fbStateSetup(stPositionState:=fbIM1K1.stOut, fPosition:=-8.82, sPmpsState:='IM1K1:PPM-OUT');
fbStateSetup(stPositionState:=fbIM1K1.stPower, fPosition:=-47.92, sPmpsState:='IM1K1:PPM-POWERMETER');
fbStateSetup(stPositionState:=fbIM1K1.stYag1, fPosition:=-71.92, sPmpsState:='IM1K1:PPM-YAG1');
fbStateSetup(stPositionState:=fbIM1K1.stYag2, fPosition:=-97.93, sPmpsState:='IM1K1:PPM-YAG2');

fbIM1K1(
    fbFFHWO := GVL.fbFastFaultOutput1,
    fbArbiter := GVL.fbArbiter1,
    stYStage := Main.M1,
    sDeviceName := 'IM1K1:PPM',
    sTransitionKey := 'IM1K1:PPM-TRANSITION',
    bEnableMotion := TRUE,
    bEnableBeamParams := TRUE,
    bEnablePositionLimits := TRUE,
    fResponsivity := 0.0624,
);

END_PROGRAM

// ---- POUs/PRG_IM2K1_PPM.TcPOU
PROGRAM PRG_IM2K1_PPM
VAR
    {attribute 'pytmc' := 'pv: IM2K1:PPM'}
    {attribute 'TcLinkTo' := '.fbGige.iIlluminatorINT := TIIB[IM2K1-EL4004]^AO Outputs Channel 1^Analog output;
                              .fbGige.bGigePower := TIIB[IM2K1-EL2004]^Channel 2^Output;
                              .fbPowerMeter.iVoltageINT := TIIB[IM2K1-EL3062]^AI Standard Channel 1^Value;
                              .fbPowerMeter.fbTempSensor.bError := TIIB[IM2K1-EL3314]^TC Inputs Channel 1^Status^Error;
                              .fbPowerMeter.fbTempSensor.bUnderrange := TIIB[IM2K1-EL3314]^TC Inputs Channel 1^Status^Underrange;
                              .fbPowerMeter.fbTempSensor.bOverrange := TIIB[IM2K1-EL3314]^TC Inputs Channel 1^Status^Overrange;
                              .fbPowerMeter.fbTempSensor.iRaw := TIIB[IM2K1-EL3314]^TC Inputs Channel 1^Value;
                              .fbYagTempSensor.bError := TIIB[IM2K1-EL3314]^TC Inputs Channel 2^Status^Error;
                              .fbYagTempSensor.bUnderrange := TIIB[IM2K1-EL3314]^TC Inputs Channel 2^Status^Underrange;
                              .fbYagTempSensor.bOverrange := TIIB[IM2K1-EL3314]^TC Inputs Channel 2^Status^Overrange;
                              .fbYagTempSensor.iRaw := TIIB[IM2K1-EL3314]^TC Inputs Channel 2^Value'}
    fbIM2K1: FB_PPM;

    fbStateSetup: FB_StateSetupHelper;
    stDefault: ST_PositionState := (
        fVelocity := 13,
        bMoveOk := TRUE,
        bValid := TRUE
    );
END_VAR


fbStateSetup(stPositionState:=stDefault, bSetDefault:=TRUE);

fbStateSetup(stPositionState:=fbIM2K1.stOut, fPosition:=-9.09, sPmpsState:='IM2K1:PPM-OUT');
fbStateSetup(stPositionState:=fbIM2K1.stPower, fPosition:=-48.19, sPmpsState:='IM2K1:PPM-POWERMETER');
fbStateSetup(stPositionState:=fbIM2K1.stYag1, fPosition:=-72.19, sPmpsState:='IM2K1:PPM-YAG1');
fbStateSetup(stPositionState:=fbIM2K1.stYag2, fPosition:=-98.2, sPmpsState:='IM2K1:PPM-YAG2');

fbIM2K1(
    fbFFHWO := GVL.fbFastFaultOutput1,
    fbArbiter := GVL.fbArbiter1,
    stYStage := Main.M2,
    sDeviceName := 'IM2K1:PPM',
    sTransitionKey := 'IM2K1:PPM-TRANSITION',
    bEnableMotion := TRUE,
    bEnableBeamParams := TRUE,
    bEnablePositionLimits := TRUE,
    fResponsivity := 0.0625,
);

END_PROGRAM

// ---- POUs/PRG_IM1K2_PPM.TcPOU
PROGRAM PRG_IM1K2_PPM
VAR
    {attribute 'pytmc' := 'pv: IM1K2:PPM'}
    {attribute 'TcLinkTo' := '.fbGige.iIlluminatorINT := TIIB[IM1K2-EL4004-E7]^AO Outputs Channel 1^Analog output;
                              .fbGige.bGigePower := TIIB[IM1K2-EL2004-E3]^Channel 2^Output;
                              .fbPowerMeter.iVoltageINT := TIIB[IM1K2-EL3062-E6]^AI Standard Channel 1^Value;
                              .fbPowerMeter.fbTempSensor.bError := TIIB[IM1K2-EL3314-E4]^TC Inputs Channel 1^Status^Error;
                              .fbPowerMeter.fbTempSensor.bUnderrange := TIIB[IM1K2-EL3314-E4]^TC Inputs Channel 1^Status^Underrange;
                              .fbPowerMeter.fbTempSensor.bOverrange := TIIB[IM1K2-EL3314-E4]^TC Inputs Channel 1^Status^Overrange;
                              .fbPowerMeter.fbTempSensor.iRaw := TIIB[IM1K2-EL3314-E4]^TC Inputs Channel 1^Value;
                              .fbYagTempSensor.bError := TIIB[IM1K2-EL3314-E4]^TC Inputs Channel 2^Status^Error;
                              .fbYagTempSensor.bUnderrange := TIIB[IM1K2-EL3314-E4]^TC Inputs Channel 2^Status^Underrange;
                              .fbYagTempSensor.bOverrange := TIIB[IM1K2-EL3314-E4]^TC Inputs Channel 2^Status^Overrange;
                              .fbYagTempSensor.iRaw := TIIB[IM1K2-EL3314-E4]^TC Inputs Channel 2^Value;
                              .fbFlowMeter.iRaw := TIIB[IM1K2-EL3052-E5]^AI Standard Channel 1^Value'}
    fbIM1K2: FB_PPM;

    fbStateSetup: FB_StateSetupHelper;
    stDefault: ST_PositionState := (
        fVelocity := 12,
        bMoveOk := TRUE,
        bValid := TRUE
    );
END_VAR


fbStateSetup(stPositionState:=stDefault, bSetDefault:=TRUE);

fbStateSetup(stPositionState:=fbIM1K2.stOut, fPosition:=-9.82, sPmpsState:='IM1K2:PPM-OUT');
fbStateSetup(stPositionState:=fbIM1K2.stPower, fPosition:=-48.92, sPmpsState:='IM1K2:PPM-POWERMETER');
fbStateSetup(stPositionState:=fbIM1K2.stYag1, fPosition:=-72.92, sPmpsState:='IM1K2:PPM-YAG1');
fbStateSetup(stPositionState:=fbIM1K2.stYag2, fPosition:=-98.93, sPmpsState:='IM1K2:PPM-YAG2');

fbIM1K2(
    fbFFHWO := GVL.fbFastFaultOutput1,
    fbArbiter := GVL.fbArbiter1,
    stYStage := Main.M4,
    sDeviceName := 'IM1K2:PPM',
    sTransitionKey := 'IM1K2:PPM-TRANSITION',
    bEnableMotion := TRUE,
    bEnableBeamParams := TRUE,
    bEnablePositionLimits := TRUE,
    fResponsivity := 0.0513,
);

END_PROGRAM

// ---- POUs/PRG_AL1K2_L2SI.TcPOU
PROGRAM PRG_AL1K2_L2SI
VAR
    {attribute 'pytmc' := 'pv: AL1K2:L2SI'}
    {attribute 'TcLinkTo' := '.fbLaser.iLaserINT := TIIB[AL1K2-EL4004-E4]^AO Outputs Channel 1^Analog output;
                              .fbLaser.iShutdownINT := TIIB[AL1K2-EL4004-E4]^AO Outputs Channel 2^Analog output'}
    fbAL1K2: FB_REF;

    fbStateSetup: FB_StateSetupHelper;
    stDefault: ST_PositionState := (
        fVelocity := 10,
        bMoveOk := TRUE,
        bValid := TRUE
    );
END_VAR


fbStateSetup(stPositionState:=stDefault, bSetDefault:=TRUE);

fbStateSetup(stPositionState:=fbAL1K2.stOut, fPosition:=-33.5, sPmpsState:='AL1K2:L2SI-OUT');
fbStateSetup(stPositionState:=fbAL1K2.stIn, fPosition:=-75, sPmpsState:='AL1K2:L2SI-IN');

fbAL1K2(
    fbFFHWO := GVL.fbFastFaultOutput2,
    fbArbiter := GVL.fbArbiter2,
    stYStage := Main.M5,
    sDeviceName := 'AL1K2:L2SI',
    sTransitionKey := 'AL1K2:L2SI-TRANSITION',
    bEnableMotion := TRUE,
    bEnableBeamParams := TRUE,
    bEnablePositionLimits := TRUE,
);

END_PROGRAM

// ---- POUs/PRG_IM2K2_PPM.TcPOU
PROGRAM PRG_IM2K2_PPM
VAR
    {attribute 'pytmc' := 'pv: IM2K2:PPM'}
    {attribute 'TcLinkTo' := '.fbGige.iIlluminatorINT := TIIB[IM2K2-EL4004-E7]^AO Outputs Channel 1^Analog output;
                              .fbGige.bGigePower := TIIB[IM2K2-EL2004-E3]^Channel 2^Output;
                              .fbPowerMeter.iVoltageINT := TIIB[IM2K2-EL3062-E6]^AI Standard Channel 1^Value;
                              .fbPowerMeter.fbTempSensor.bError := TIIB[IM2K2-EL3314-E4]^TC Inputs Channel 1^Status^Error;
                              .fbPowerMeter.fbTempSensor.bUnderrange := TIIB[IM2K2-EL3314-E4]^TC Inputs Channel 1^Status^Underrange;
                              .fbPowerMeter.fbTempSensor.bOverrange := TIIB[IM2K2-EL3314-E4]^TC Inputs Channel 1^Status^Overrange;
                              .fbPowerMeter.fbTempSensor.iRaw := TIIB[IM2K2-EL3314-E4]^TC Inputs Channel 1^Value;
                              .fbYagTempSensor.bError := TIIB[IM2K2-EL3314-E4]^TC Inputs Channel 2^Status^Error;
                              .fbYagTempSensor.bUnderrange := TIIB[IM2K2-EL3314-E4]^TC Inputs Channel 2^Status^Underrange;
                              .fbYagTempSensor.bOverrange := TIIB[IM2K2-EL3314-E4]^TC Inputs Channel 2^Status^Overrange;
                              .fbYagTempSensor.iRaw := TIIB[IM2K2-EL3314-E4]^TC Inputs Channel 2^Value;
                              .fbFlowMeter.iRaw := TIIB[IM1K2-EL3052-E5]^AI Standard Channel 1^Value'}
// IM2K2 shares the same flow meter as IM1K2
    fbIM2K2: FB_PPM;

    fbStateSetup: FB_StateSetupHelper;
    stDefault: ST_PositionState := (
        fVelocity := 15,
        bMoveOk := TRUE,
        bValid := TRUE
    );
END_VAR


fbStateSetup(stPositionState:=stDefault, bSetDefault:=TRUE);

fbStateSetup(stPositionState:=fbIM2K2.stOut, fPosition:=-8.49, sPmpsState:='IM2K2:PPM-OUT');
fbStateSetup(stPositionState:=fbIM2K2.stPower, fPosition:=-47.59, sPmpsState:='IM2K2:PPM-POWERMETER');
fbStateSetup(stPositionState:=fbIM2K2.stYag1, fPosition:=-71.59, sPmpsState:='IM2K2:PPM-YAG1');
fbStateSetup(stPositionState:=fbIM2K2.stYag2, fPosition:=-97.60, sPmpsState:='IM2K2:PPM-YAG2');

fbIM2K2(
    fbFFHWO := GVL.fbFastFaultOutput2,
    fbArbiter := GVL.fbArbiter2,
    stYStage := Main.M6,
    sDeviceName := 'IM2K2:PPM',
    sTransitionKey := 'IM2K2:PPM-TRANSITION',
    bEnableMotion := TRUE,
    bEnableBeamParams := TRUE,
    bEnablePositionLimits := TRUE,
    fResponsivity := 0.0670,
);

END_PROGRAM

// ---- POUs/PRG_IM3K2_PPM.TcPOU
PROGRAM PRG_IM3K2_PPM
VAR
    {attribute 'pytmc' := 'pv: IM3K2:PPM'}
    {attribute 'TcLinkTo' := '.fbGige.iIlluminatorINT := TIIB[IM3K2-EL4004-E7]^AO Outputs Channel 1^Analog output;
                              .fbGige.bGigePower := TIIB[IM3K2-EL2004-E3]^Channel 2^Output;
                              .fbPowerMeter.iVoltageINT := TIIB[IM3K2-EL3062-E6]^AI Standard Channel 1^Value;
                              .fbPowerMeter.fbTempSensor.bError := TIIB[IM3K2-EL3314-E4]^TC Inputs Channel 1^Status^Error;
                              .fbPowerMeter.fbTempSensor.bUnderrange := TIIB[IM3K2-EL3314-E4]^TC Inputs Channel 1^Status^Underrange;
                              .fbPowerMeter.fbTempSensor.bOverrange := TIIB[IM3K2-EL3314-E4]^TC Inputs Channel 1^Status^Overrange;
                              .fbPowerMeter.fbTempSensor.iRaw := TIIB[IM3K2-EL3314-E4]^TC Inputs Channel 1^Value;
                              .fbYagTempSensor.bError := TIIB[IM3K2-EL3314-E4]^TC Inputs Channel 2^Status^Error;
                              .fbYagTempSensor.bUnderrange := TIIB[IM3K2-EL3314-E4]^TC Inputs Channel 2^Status^Underrange;
                              .fbYagTempSensor.bOverrange := TIIB[IM3K2-EL3314-E4]^TC Inputs Channel 2^Status^Overrange;
                              .fbYagTempSensor.iRaw := TIIB[IM3K2-EL3314-E4]^TC Inputs Channel 2^Value;
                              .fbFlowMeter.iRaw := TIIB[IM1K2-EL3052-E5]^AI Standard Channel 1^Value'}
// IM3K2 shares the same flow meter as IM1K2
    fbIM3K2: FB_PPM;

    fbStateSetup: FB_StateSetupHelper;
    stDefault: ST_PositionState := (
        fVelocity := 14,
        bMoveOk := TRUE,
        bValid := TRUE
    );
END_VAR


fbStateSetup(stPositionState:=stDefault, bSetDefault:=TRUE);

fbStateSetup(stPositionState:=fbIM3K2.stOut, fPosition:=-9.61, sPmpsState:='IM3K2:PPM-OUT');
fbStateSetup(stPositionState:=fbIM3K2.stPower, fPosition:=-48.71, sPmpsState:='IM3K2:PPM-POWERMETER');
fbStateSetup(stPositionState:=fbIM3K2.stYag1, fPosition:=-72.71, sPmpsState:='IM3K2:PPM-YAG1');
fbStateSetup(stPositionState:=fbIM3K2.stYag2, fPosition:=-98.72, sPmpsState:='IM3K2:PPM-YAG2');

fbIM3K2(
    fbFFHWO := GVL.fbFastFaultOutput2,
    fbArbiter := GVL.fbArbiter2,
    stYStage := Main.M7,
    sDeviceName := 'IM3K2:PPM',
    sTransitionKey := 'IM3K2:PPM-TRANSITION',
    bEnableMotion := TRUE,
    bEnableBeamParams := TRUE,
    bEnablePositionLimits := TRUE,
    fResponsivity := 0.0503
);

END_PROGRAM

// ---- POUs/PRG_IM4K2_PPM.TcPOU
PROGRAM PRG_IM4K2_PPM
VAR
    {attribute 'pytmc' := 'pv: IM4K2:PPM'}
    {attribute 'TcLinkTo' := '.fbGige.iIlluminatorINT := TIIB[IM4K2-EL4004-E7]^AO Outputs Channel 1^Analog output;
                              .fbGige.bGigePower := TIIB[IM4K2-EL2004-E3]^Channel 2^Output;
                              .fbPowerMeter.iVoltageINT := TIIB[IM4K2-EL3602-0002-E8]^AI Inputs Channel 1^Value;
                              .fbPowerMeter.fbTempSensor.bError := TIIB[IM4K2-EL3314-E4]^TC Inputs Channel 1^Status^Error;
                              .fbPowerMeter.fbTempSensor.bUnderrange := TIIB[IM4K2-EL3314-E4]^TC Inputs Channel 1^Status^Underrange;
                              .fbPowerMeter.fbTempSensor.bOverrange := TIIB[IM4K2-EL3314-E4]^TC Inputs Channel 1^Status^Overrange;
                              .fbPowerMeter.fbTempSensor.iRaw := TIIB[IM4K2-EL3314-E4]^TC Inputs Channel 1^Value;
                              .fbYagTempSensor.bError := TIIB[IM4K2-EL3314-E4]^TC Inputs Channel 2^Status^Error;
                              .fbYagTempSensor.bUnderrange := TIIB[IM4K2-EL3314-E4]^TC Inputs Channel 2^Status^Underrange;
                              .fbYagTempSensor.bOverrange := TIIB[IM4K2-EL3314-E4]^TC Inputs Channel 2^Status^Overrange;
                              .fbYagTempSensor.iRaw := TIIB[IM4K2-EL3314-E4]^TC Inputs Channel 2^Value;
                              .fbFlowMeter.iRaw := TIIB[IM1K2-EL3052-E5]^AI Standard Channel 1^Value'}
// IM4K2 shares the same flow meter as IM1K2
    fbIM4K2: FB_PPM;

    fbStateSetup: FB_StateSetupHelper;
    stDefault: ST_PositionState := (
        fVelocity := 12,
        bMoveOk := TRUE,
        bValid := TRUE
    );
END_VAR


fbStateSetup(stPositionState:=stDefault, bSetDefault:=TRUE);

fbStateSetup(stPositionState:=fbIM4K2.stOut, fPosition:=-10.80, sPmpsState:='IM4K2:PPM-OUT');
fbStateSetup(stPositionState:=fbIM4K2.stPower, fPosition:=-49.90, sPmpsState:='IM4K2:PPM-POWERMETER');
fbStateSetup(stPositionState:=fbIM4K2.stYag1, fPosition:=-73.90, sPmpsState:='IM4K2:PPM-YAG1');
fbStateSetup(stPositionState:=fbIM4K2.stYag2, fPosition:=-99.91, sPmpsState:='IM4K2:PPM-YAG2');

fbIM4K2(
    fbFFHWO := GVL.fbFastFaultOutput2,
    fbArbiter := GVL.fbArbiter2,
    stYStage := Main.M8,
    sDeviceName := 'IM4K2:PPM',
    sTransitionKey := 'IM4K2:PPM-TRANSITION',
    bEnableMotion := TRUE,
    bEnableBeamParams := TRUE,
    bEnablePositionLimits := TRUE,
    fResponsivity := 0.0584,
    iTermBits := 31,
    fTermMax := 200,
    fTermMin := 0,
);

END_PROGRAM

// ---- POUs/PRG_TM1K2_ATM.TcPOU
PROGRAM PRG_TM1K2_ATM
VAR
    {attribute 'pytmc' := 'pv: TM1K2:ATM'}
    {attribute 'TcLinkTo' := '.fbThermoCouple1.bError := TIIB[TM1K2-EL3314-E5]^TC Inputs Channel 1^Status^Error;
                              .fbThermoCouple1.bUnderrange := TIIB[TM1K2-EL3314-E5]^TC Inputs Channel 1^Status^Underrange;
                              .fbThermoCouple1.bOverrange := TIIB[TM1K2-EL3314-E5]^TC Inputs Channel 1^Status^Overrange;
                              .fbThermoCouple1.iRaw := TIIB[TM1K2-EL3314-E5]^TC Inputs Channel 1^Value;
                              .fbFlowMeter.iRaw := TIIB[AT1K2-EL3052-E8]^AI Standard Channel 1^Value

'} // TM1K2 shares the same cooling meter as AT1K2
    fbTM1K2: FB_TM1K2;

    fbStateSetup: FB_StateSetupHelper;
    stDefault: ST_PositionState := (
        fVelocity := 1,
        bMoveOk := TRUE,
        bValid := TRUE
    );
END_VAR


fbStateSetup(stPositionState:=stDefault, bSetDefault:=TRUE);

fbStateSetup(stPositionState:=fbTM1K2.stOut, fPosition:=-16.00, fDelta:=7, sPmpsState:='TM1K2:ATM-OUT');
fbStateSetup(stPositionState:=fbTM1K2.stTarget1, fPosition:=-28, fDelta:=7, sPmpsState:='TM1K2:ATM-TARGET1');
fbStateSetup(stPositionState:=fbTM1K2.stTarget2, fPosition:=-38, fDelta:=7, sPmpsState:='TM1K2:ATM-TARGET2');
fbStateSetup(stPositionState:=fbTM1K2.stTarget3, fPosition:=-48, fDelta:=7, sPmpsState:='TM1K2:ATM-TARGET3');
fbStateSetup(stPositionState:=fbTM1K2.stTarget4, fPosition:=-58, fDelta:=7, sPmpsState:='TM1K2:ATM-TARGET4');
fbStateSetup(stPositionState:=fbTM1K2.stTarget5, fPosition:=-68, fDelta:=7, sPmpsState:='TM1K2:ATM-TARGET5');
fbStateSetup(stPositionState:=fbTM1K2.stTarget6, fPosition:=-80, fDelta:=7, sPmpsState:='TM1K2:ATM-TARGET6');
fbStateSetup(stPositionState:=fbTM1K2.stTarget7, fPosition:=-96, fDelta:=7, sPmpsState:='TM1K2:ATM-TARGET7');
fbStateSetup(stPositionState:=fbTM1K2.stTarget8, fPosition:=-114.5, fDelta:=7, sPmpsState:='TM1K2:ATM-TARGET8');

fbTM1K2(
    fbFFHWO := GVL.fbFastFaultOutput2,
    fbArbiter := GVL.fbArbiter2,
    stYStage := Main.M9,
    stXStage := Main.M10,
    sDeviceName := 'TM1K2:ATM',
    sTransitionKey := 'TM1K2:ATM-TRANSITION',
    bEnableMotion := TRUE,
    bEnableBeamParams := TRUE,
    bEnablePositionLimits := TRUE,
);

END_PROGRAM

// ---- POUs/TM1K2/FB_TM1K2.TcPOU
FUNCTION_BLOCK FB_TM1K2
(*
    Function block for Arrival Time Monitor (ATM) controls:
    - X, Y motion
    - Y target states
    - thermocouple

    For TM1K2, we make the following adjustments:
    - Add stTarget6 to the inputs
    - Change the array pragma from 1..6 to 1..7 (1 out and 6 in states, up from 5 in states)
    - Use E_TM1K2_States instead of E_ATM_States

    Add array to 1..9
*)
VAR_IN_OUT
    // Y motor (state select).
    stYStage: ST_MotionStage;
    // X motor (align target to beam).
    stXStage: ST_MotionStage;
    // The fast fault output to fault to.
    fbFFHWO: FB_HardwareFFOutput;
    // The arbiter to request beam conditions from.
    fbArbiter: FB_Arbiter;
END_VAR
VAR_INPUT
    // Settings for the OUT state.
    stOut: ST_PositionState;
    // Settings for the TARGET1 state.
    stTarget1: ST_PositionState;
    // Settings for the TARGET2 state.
    stTarget2: ST_PositionState;
    // Settings for the TARGET3 state.
    stTarget3: ST_PositionState;
    // Settings for the TARGET4 state.
    stTarget4: ST_PositionState;
    // Settings for the TARGET5 state.
    stTarget5: ST_PositionState;
    // Settings for the TARGET6 state.
    stTarget6: ST_PositionState;
    // Settings for the TARGET7 state.
    stTarget7: ST_PositionState;
    // Settings for the TARGET8 state.
    stTarget8: ST_PositionState;
    // Set this to a non-unknown value to request a new move.
    {attribute 'pytmc' := '
        pv: MMS:STATE:SET
        io: io
    '}
    eEnumSet: E_TM1K2_States;
    // Set this to TRUE to enable input state moves, or FALSE to disable them.
    bEnableMotion: BOOL;
    // Set this to TRUE to enable beam parameter checks, or FALSE to disable them.
    bEnableBeamParams: BOOL;
    // Set this to TRUE to enable position limit checks, or FALSE to disable them.
    bEnablePositionLimits: BOOL;
    // The name of the device for use in the PMPS DB lookup and diagnostic screens.
    sDeviceName: STRING;
    // The name of the transition state in the PMPS database.
    sTransitionKey: STRING;
    // Set this to TRUE to re-read the loaded database immediately (useful for debug).
    bReadDBNow: BOOL;
END_VAR
VAR_OUTPUT
    // The current position state as an enum.
    {attribute 'pytmc' := '
        pv: MMS:STATE:GET
        io: i
    '}
    eEnumGet: E_TM1K2_States;
    // The PMPS database lookup associated with the current position state.
    stDbStateParams: ST_DbStateParams;
END_VAR
VAR
    bInit: BOOL;

    fbYStage: FB_MotionStage;
    fbXStage: FB_MotionStage;

    fbStateDefaults: FB_PositionState_Defaults;

    {attribute 'pytmc' := '
        pv: MMS
        astPositionState.array: 1..7
    '}
    fbStates: FB_PositionStatePMPS1D;
    astPositionState: ARRAY[1..GeneralConstants.MAX_STATES] OF ST_PositionState;
    fbArrCheckWrite: FB_CheckPositionStateWrite;

    {attribute 'pytmc' := 'pv: STC:01'}
    fbThermoCouple1: FB_TempSensor;

    {attribute 'pytmc' :='pv: FWM'}
    fbFlowMeter: FB_AnalogInput := (iTermBits:=15, fTermMax:=60, fTermMin:=0);
END_VAR
VAR CONSTANT
    // State defaults if not provided
    fDelta: LREAL := 2;
    fAccel: LREAL := 200;
    fOutDecel: LREAL := 25;
END_VAR


IF NOT bInit THEN
    bInit := TRUE;

    stYStage.nEnableMode := E_StageEnableMode.DURING_MOTION;
    stXStage.nEnableMode := E_StageEnableMode.DURING_MOTION;

    // Partial backcompat, this used to set fVelocity too but this should be set per install
    fbStateDefaults(stPositionState:=stOut, sNameDefault:='OUT', fDeltaDefault:=fDelta, fAccelDefault:=fAccel, fDecelDefault:=fOutDecel);
    fbStateDefaults(stPositionState:=stTarget1, sNameDefault:='TARGET1', fDeltaDefault:=fDelta, fAccelDefault:=fAccel, fDecelDefault:=fAccel);
    fbStateDefaults(stPositionState:=stTarget2, sNameDefault:='TARGET2', fDeltaDefault:=fDelta, fAccelDefault:=fAccel, fDecelDefault:=fAccel);
    fbStateDefaults(stPositionState:=stTarget3, sNameDefault:='TARGET3', fDeltaDefault:=fDelta, fAccelDefault:=fAccel, fDecelDefault:=fAccel);
    fbStateDefaults(stPositionState:=stTarget4, sNameDefault:='TARGET4', fDeltaDefault:=fDelta, fAccelDefault:=fAccel, fDecelDefault:=fAccel);
    fbStateDefaults(stPositionState:=stTarget5, sNameDefault:='TARGET5', fDeltaDefault:=fDelta, fAccelDefault:=fAccel, fDecelDefault:=fAccel);
    fbStateDefaults(stPositionState:=stTarget6, sNameDefault:='TARGET6', fDeltaDefault:=fDelta, fAccelDefault:=fAccel, fDecelDefault:=fAccel);
    fbStateDefaults(stPositionState:=stTarget7, sNameDefault:='TARGET7', fDeltaDefault:=fDelta, fAccelDefault:=fAccel, fDecelDefault:=fAccel);
    fbStateDefaults(stPositionState:=stTarget8, sNameDefault:='TARGET8', fDeltaDefault:=fDelta, fAccelDefault:=fAccel, fDecelDefault:=fAccel);
END_IF

stYStage.bHardwareEnable := TRUE;
stYStage.bPowerSelf := FALSE;

stXStage.bLimitForwardEnable := TRUE;
stXStage.bLimitBackwardEnable := TRUE;
stXStage.bHardwareEnable := TRUE;
stXStage.bPowerSelf := TRUE;

fbYStage(stMotionStage:=stYStage);
fbXStage(stMotionStage:=stXStage);

// We need to update from PLC or from EPICS, but not both
fbArrCheckWrite(
    astPositionState:=astPositionState,
    bCheck:=TRUE,
    bSave:=FALSE,
);
IF NOT fbArrCheckWrite.bHadWrite THEN
    astPositionState[E_TM1K2_States.OUT] := stOut;
    astPositionState[E_TM1K2_States.TARGET1] := stTarget1;
    astPositionState[E_TM1K2_States.TARGET2] := stTarget2;
    astPositionState[E_TM1K2_States.TARGET3] := stTarget3;
    astPositionState[E_TM1K2_States.TARGET4] := stTarget4;
    astPositionState[E_TM1K2_States.TARGET5] := stTarget5;
    astPositionState[E_TM1K2_States.TARGET6] := stTarget6;
    astPositionState[E_TM1K2_States.TARGET7] := stTarget7;
    astPositionState[E_TM1K2_States.TARGET8] := stTarget8;
END_IF

fbStates(
    stMotionStage:=stYStage,
    astPositionState:=astPositionState,
    eEnumSet:=eEnumSet,
    eEnumGet:=eEnumGet,
    fbFFHWO:=fbFFHWO,
    fbArbiter:=fbArbiter,
    bEnableMotion:=bEnableMotion,
    bEnableBeamParams:=bEnableBeamParams,
    bEnablePositionLimits:=bEnablePositionLimits,
    sDeviceName:=sDeviceName,
    sTransitionKey:=sTransitionKey,
    bReadDBNow:=bReadDBNow,
    stDbStateParams=>stDbStateParams,
);

fbArrCheckWrite(
    astPositionState:=astPositionState,
    bCheck:=FALSE,
    bSave:=TRUE,
);

stOut := astPositionState[E_TM1K2_States.OUT];
stTarget1 := astPositionState[E_TM1K2_States.TARGET1];
stTarget2 := astPositionState[E_TM1K2_States.TARGET2];
stTarget3 := astPositionState[E_TM1K2_States.TARGET3];
stTarget4 := astPositionState[E_TM1K2_States.TARGET4];
stTarget5 := astPositionState[E_TM1K2_States.TARGET5];
stTarget6 := astPositionState[E_TM1K2_States.TARGET6];
stTarget7 := astPositionState[E_TM1K2_States.TARGET7];
stTarget8 := astPositionState[E_TM1K2_States.TARGET8];

fbThermoCouple1();
fbFlowMeter();

END_FUNCTION_BLOCK

// ---- POUs/PRG_LI2K2_K2A.TcPOU
PROGRAM PRG_LI2K2_K2A
VAR
    {attribute 'pytmc' := 'pv: LI2K2:K2A'}
    fbLI2K2: FB_LIC;

    fbStateSetup: FB_StateSetupHelper;
    stDefault: ST_PositionState := (
        fVelocity := 1,
        bMoveOk := TRUE,
        bValid := TRUE
    );
END_VAR


fbStateSetup(stPositionState:=stDefault, bSetDefault:=TRUE);

fbStateSetup(stPositionState:=fbLI2K2.stOut, fPosition:=1.2, sPmpsState:='LI2K2:K2A-OUT');
fbStateSetup(stPositionState:=fbLI2K2.stMirror1, fPosition:=-35.3, sPmpsState:='LI2K2:K2A-MIRROR1');
fbStateSetup(stPositionState:=fbLI2K2.stMirror2, fPosition:=-69.3, sPmpsState:='LI2K2:K2A-MIRROR2');
fbStateSetup(stPositionState:=fbLI2K2.stTarget1, fPosition:=-101.3, sPmpsState:='LI2K2:K2A-TARGET1');

fbLI2K2(
    fbFFHWO := GVL.fbFastFaultOutput2,
    fbArbiter := GVL.fbArbiter2,
    stYStage := Main.M11,
    sDeviceName := 'LI2K2:K2A',
    sTransitionKey := 'LI2K2:K2A-TRANSITION',
    bEnableMotion := TRUE,
    bEnableBeamParams := TRUE,
    bEnablePositionLimits := TRUE,
);

END_PROGRAM

// ---- POUs/PRG_PF1K2_WFS.TcPOU
PROGRAM PRG_PF1K2_WFS
VAR
    {attribute 'pytmc' := 'pv: PF1K2:WFS'}
    {attribute 'TcLinkTo' := '.fbThermoCouple1.bError 		:= TIIB[PF1K2-EL3314-E5]^TC Inputs Channel 1^Status^Error;
                              .fbThermoCouple1.bUnderrange	:= TIIB[PF1K2-EL3314-E5]^TC Inputs Channel 1^Status^Underrange;
                              .fbThermoCouple1.bOverrange 	:= TIIB[PF1K2-EL3314-E5]^TC Inputs Channel 1^Status^Overrange;
                              .fbThermoCouple1.iRaw 		:= TIIB[PF1K2-EL3314-E5]^TC Inputs Channel 1^Value;
                              .fbThermoCouple2.bError 		:= TIIB[PF1K2-EL3314-E5]^TC Inputs Channel 2^Status^Error;
                              .fbThermoCouple2.bUnderrange 	:= TIIB[PF1K2-EL3314-E5]^TC Inputs Channel 2^Status^Underrange;
                              .fbThermoCouple2.bOverrange 	:= TIIB[PF1K2-EL3314-E5]^TC Inputs Channel 2^Status^Overrange;
                              .fbThermoCouple2.iRaw 		:= TIIB[PF1K2-EL3314-E5]^TC Inputs Channel 2^Value;
                              .fbFlowMeter.iRaw := TIIB[IM5K2-EL3052-E5]^AI Standard Channel 1^Value

'} // PF1K2 shares the same flow meter as IM5K2
    fbPF1K2: FB_WFS;

    fbStateSetup: FB_StateSetupHelper;
    stDefault: ST_PositionState := (
        fVelocity := 1,
        bMoveOk := TRUE,
        bValid := TRUE
    );
END_VAR


fbStateSetup(stPositionState:=stDefault, bSetDefault:=TRUE);

fbStateSetup(stPositionState:=fbPF1K2.stOut, fPosition:=-13.80, sPmpsState:='PF1K2:WFS-OUT');
fbStateSetup(stPositionState:=fbPF1K2.stTarget1, fPosition:=-94.00, sPmpsState:='PF1K2:WFS-TARGET1');
fbStateSetup(stPositionState:=fbPF1K2.stTarget2, fPosition:=-82.755, sPmpsState:='PF1K2:WFS-TARGET2');
fbStateSetup(stPositionState:=fbPF1K2.stTarget3, fPosition:=-68.38, sPmpsState:='PF1K2:WFS-TARGET3');
fbStateSetup(stPositionState:=fbPF1K2.stTarget4, fPosition:=-54.004, sPmpsState:='PF1K2:WFS-TARGET4');
fbStateSetup(stPositionState:=fbPF1K2.stTarget5, fPosition:=-39.629, sPmpsState:='PF1K2:WFS-TARGET5');

fbPF1K2(
    fbFFHWO := GVL.fbFastFaultOutput2,
    fbArbiter := GVL.fbArbiter2,
    stYStage := Main.M12,
    stZStage := Main.M13,
    sDeviceName := 'PF1K2:WFS',
    sTransitionKey := 'PF1K2:WFS-TRANSITION',
    bEnableMotion := TRUE,
    bEnableBeamParams := TRUE,
    bEnablePositionLimits := TRUE,
    eEnumGet=>GVL.ePF1K2State,
);

END_PROGRAM

// ---- POUs/PRG_IM5K2_PPM.TcPOU
PROGRAM PRG_IM5K2_PPM
VAR
    {attribute 'pytmc' := 'pv: IM5K2:PPM'}
    {attribute 'TcLinkTo' := '.fbGige.iIlluminatorINT := TIIB[IM5K2-EL4004-E7]^AO Outputs Channel 1^Analog output;
                              .fbGige.bGigePower := TIIB[IM5K2-EL2004-E3]^Channel 2^Output;
                              .fbPowerMeter.iVoltageINT := TIIB[IM5K2-EL3062-E6]^AI Standard Channel 1^Value;
                              .fbPowerMeter.fbTempSensor.bError := TIIB[IM5K2-EL3314-E4]^TC Inputs Channel 1^Status^Error;
                              .fbPowerMeter.fbTempSensor.bUnderrange := TIIB[IM5K2-EL3314-E4]^TC Inputs Channel 1^Status^Underrange;
                              .fbPowerMeter.fbTempSensor.bOverrange := TIIB[IM5K2-EL3314-E4]^TC Inputs Channel 1^Status^Overrange;
                              .fbPowerMeter.fbTempSensor.iRaw := TIIB[IM5K2-EL3314-E4]^TC Inputs Channel 1^Value;
                              .fbYagTempSensor.bError := TIIB[IM5K2-EL3314-E4]^TC Inputs Channel 2^Status^Error;
                              .fbYagTempSensor.bUnderrange := TIIB[IM5K2-EL3314-E4]^TC Inputs Channel 2^Status^Underrange;
                              .fbYagTempSensor.bOverrange := TIIB[IM5K2-EL3314-E4]^TC Inputs Channel 2^Status^Overrange;
                              .fbYagTempSensor.iRaw := TIIB[IM5K2-EL3314-E4]^TC Inputs Channel 2^Value;
                              .fbFlowMeter.iRaw := TIIB[IM5K2-EL3052-E5]^AI Standard Channel 1^Value'}
    fbIM5K2: FB_PPM;

    fbStateSetup: FB_StateSetupHelper;
    stDefault: ST_PositionState := (
        fVelocity := 12,
        bMoveOk := TRUE,
        bValid := TRUE
    );
END_VAR


fbStateSetup(stPositionState:=stDefault, bSetDefault:=TRUE);

fbStateSetup(stPositionState:=fbIM5K2.stOut, fPosition:=-8.92, sPmpsState:='IM5K2:PPM-OUT');
fbStateSetup(stPositionState:=fbIM5K2.stPower, fPosition:=-48.02, sPmpsState:='IM5K2:PPM-POWERMETER');
fbStateSetup(stPositionState:=fbIM5K2.stYag1, fPosition:=-72.02);
fbStateSetup(stPositionState:=fbIM5K2.stYag2, fPosition:=-98.03, sPmpsState:='IM5K2:PPM-YAG2');

CASE GVL.ePF1K2State OF
    E_WFS_STATES.TARGET1, E_WFS_STATES.TARGET2, E_WFS_STATES.TARGET3, E_WFS_STATES.TARGET4, E_WFS_STATES.TARGET5 :
        // Known state targets: allow less strict pmps
        fbIM5K2.stYag1.stPMPS.sPmpsState := 'IM5K2:PPM-YAG1_WFS_IN';
ELSE
    // Out, Unknown, or an unexpected state: full pmps
    fbIM5K2.stYag1.stPMPS.sPmpsState := 'IM5K2:PPM-YAG1';
END_CASE

fbIM5K2(
    fbFFHWO := GVL.fbFastFaultOutput2,
    fbArbiter := GVL.fbArbiter2,
    stYStage := Main.M14,
    sDeviceName := 'IM5K2:PPM',
    sTransitionKey := 'IM5K2:PPM-TRANSITION',
    bEnableMotion := TRUE,
    bEnableBeamParams := TRUE,
    bEnablePositionLimits := TRUE,
    fResponsivity := 0.0574,
);

END_PROGRAM

// ---- POUs/PRG_TM2K2_ATM.TcPOU
PROGRAM PRG_TM2K2_ATM
VAR
    {attribute 'pytmc' := 'pv: TM2K2:ATM'}
    {attribute 'TcLinkTo' := '.fbThermoCouple1.bError := TIIB[TM2K2-EL3314-E5]^TC Inputs Channel 1^Status^Error;
                              .fbThermoCouple1.bUnderrange := TIIB[TM2K2-EL3314-E5]^TC Inputs Channel 1^Status^Underrange;
                              .fbThermoCouple1.bOverrange := TIIB[TM2K2-EL3314-E5]^TC Inputs Channel 1^Status^Overrange;
                              .fbThermoCouple1.iRaw := TIIB[TM2K2-EL3314-E5]^TC Inputs Channel 1^Value;
                              .fbFlowMeter.iRaw := TIIB[TM2K2-EL3052-E6]^AI Standard Channel 1^Value
'}
    fbTM2K2: FB_TM2K2;

    fbStateSetup: FB_StateSetupHelper;
    stDefault: ST_PositionState := (
        fVelocity := 1,
        bMoveOk := TRUE,
        bValid := TRUE
    );
END_VAR


fbStateSetup(stPositionState:=stDefault, bSetDefault:=TRUE);

fbStateSetup(stPositionState:=fbTM2K2.stOut, fPosition:=5.3, fDelta:=7, sPmpsState:='TM2K2:ATM-OUT');
fbStateSetup(stPositionState:=fbTM2K2.stTarget1, fPosition:=-15.5, fDelta:=7, sPmpsState:='TM2K2:ATM-TARGET1');
fbStateSetup(stPositionState:=fbTM2K2.stTarget2, fPosition:=-36.5, fDelta:=7, sPmpsState:='TM2K2:ATM-TARGET2');
fbStateSetup(stPositionState:=fbTM2K2.stTarget3, fPosition:=-52.0, fDelta:=7, sPmpsState:='TM2K2:ATM-TARGET3');
fbStateSetup(stPositionState:=fbTM2K2.stTarget4, fPosition:=-61.50, fDelta:=7, sPmpsState:='TM2K2:ATM-TARGET4');
fbStateSetup(stPositionState:=fbTM2K2.stTarget5, fPosition:=-77.0, fDelta:=7, sPmpsState:='TM2K2:ATM-TARGET5');
fbStateSetup(stPositionState:=fbTM2K2.stTarget6, fPosition:=-96.6, fDelta:=7, sPmpsState:='TM2K2:ATM-TARGET6');

fbTM2K2(
    fbFFHWO := GVL.fbFastFaultOutput2,
    fbArbiter := GVL.fbArbiter2,
    stYStage := Main.M15,
    stXStage := Main.M16,
    sDeviceName := 'TM2K2:ATM',
    sTransitionKey := 'TM2K2:ATM-TRANSITION',
    bEnableMotion := TRUE,
    bEnableBeamParams := TRUE,
    bEnablePositionLimits := TRUE,
);

END_PROGRAM

// ---- POUs/TM2K2/FB_TM2K2.TcPOU
FUNCTION_BLOCK FB_TM2K2
(*
    Function block for Arrival Time Monitor (ATM) controls:
    - X, Y motion
    - Y target states
    - thermocouple

    For TM2K2, we make the following adjustments:
    - Add stTarget6 to the inputs
    - Change the array pragma from 1..6 to 1..7 (1 out and 6 in states, up from 5 in states)
    - Use E_TM2K2_States instead of E_ATM_States
*)
VAR_IN_OUT
    // Y motor (state select).
    stYStage: ST_MotionStage;
    // X motor (align target to beam).
    stXStage: ST_MotionStage;
    // The fast fault output to fault to.
    fbFFHWO: FB_HardwareFFOutput;
    // The arbiter to request beam conditions from.
    fbArbiter: FB_Arbiter;
END_VAR
VAR_INPUT
    // Settings for the OUT state.
    stOut: ST_PositionState;
    // Settings for the TARGET1 state.
    stTarget1: ST_PositionState;
    // Settings for the TARGET2 state.
    stTarget2: ST_PositionState;
    // Settings for the TARGET3 state.
    stTarget3: ST_PositionState;
    // Settings for the TARGET4 state.
    stTarget4: ST_PositionState;
    // Settings for the TARGET5 state.
    stTarget5: ST_PositionState;
    // Settings for the TARGET6 state.
    stTarget6: ST_PositionState;
    // Set this to a non-unknown value to request a new move.
    {attribute 'pytmc' := '
        pv: MMS:STATE:SET
        io: io
    '}
    eEnumSet: E_TM2K2_States;
    // Set this to TRUE to enable input state moves, or FALSE to disable them.
    bEnableMotion: BOOL;
    // Set this to TRUE to enable beam parameter checks, or FALSE to disable them.
    bEnableBeamParams: BOOL;
    // Set this to TRUE to enable position limit checks, or FALSE to disable them.
    bEnablePositionLimits: BOOL;
    // The name of the device for use in the PMPS DB lookup and diagnostic screens.
    sDeviceName: STRING;
    // The name of the transition state in the PMPS database.
    sTransitionKey: STRING;
    // Set this to TRUE to re-read the loaded database immediately (useful for debug).
    bReadDBNow: BOOL;
END_VAR
VAR_OUTPUT
    // The current position state as an enum.
    {attribute 'pytmc' := '
        pv: MMS:STATE:GET
        io: i
    '}
    eEnumGet: E_TM2K2_States;
    // The PMPS database lookup associated with the current position state.
    stDbStateParams: ST_DbStateParams;
END_VAR
VAR
    bInit: BOOL;

    fbYStage: FB_MotionStage;
    fbXStage: FB_MotionStage;

    fbStateDefaults: FB_PositionState_Defaults;

    {attribute 'pytmc' := '
        pv: MMS
        astPositionState.array: 1..7
    '}
    fbStates: FB_PositionStatePMPS1D;
    astPositionState: ARRAY[1..GeneralConstants.MAX_STATES] OF ST_PositionState;
    fbArrCheckWrite: FB_CheckPositionStateWrite;

    {attribute 'pytmc' := 'pv: STC:01'}
    fbThermoCouple1: FB_TempSensor;

    {attribute 'pytmc' :='pv: FWM'}
    fbFlowMeter: FB_AnalogInput := (iTermBits:=15, fTermMax:=60, fTermMin:=0);
END_VAR
VAR CONSTANT
    // State defaults if not provided
    fDelta: LREAL := 2;
    fAccel: LREAL := 200;
    fOutDecel: LREAL := 25;
END_VAR


IF NOT bInit THEN
    bInit := TRUE;

    stYStage.nEnableMode := E_StageEnableMode.DURING_MOTION;
    stXStage.nEnableMode := E_StageEnableMode.DURING_MOTION;

    // Partial backcompat, this used to set fVelocity too but this should be set per install
    fbStateDefaults(stPositionState:=stOut, sNameDefault:='OUT', fDeltaDefault:=fDelta, fAccelDefault:=fAccel, fDecelDefault:=fOutDecel);
    fbStateDefaults(stPositionState:=stTarget1, sNameDefault:='TARGET1', fDeltaDefault:=fDelta, fAccelDefault:=fAccel, fDecelDefault:=fAccel);
    fbStateDefaults(stPositionState:=stTarget2, sNameDefault:='TARGET2', fDeltaDefault:=fDelta, fAccelDefault:=fAccel, fDecelDefault:=fAccel);
    fbStateDefaults(stPositionState:=stTarget3, sNameDefault:='TARGET3', fDeltaDefault:=fDelta, fAccelDefault:=fAccel, fDecelDefault:=fAccel);
    fbStateDefaults(stPositionState:=stTarget4, sNameDefault:='TARGET4', fDeltaDefault:=fDelta, fAccelDefault:=fAccel, fDecelDefault:=fAccel);
    fbStateDefaults(stPositionState:=stTarget5, sNameDefault:='TARGET5', fDeltaDefault:=fDelta, fAccelDefault:=fAccel, fDecelDefault:=fAccel);
    fbStateDefaults(stPositionState:=stTarget6, sNameDefault:='TARGET6', fDeltaDefault:=fDelta, fAccelDefault:=fAccel, fDecelDefault:=fAccel);
END_IF

stYStage.bHardwareEnable := TRUE;
stYStage.bPowerSelf := FALSE;

stXStage.bLimitForwardEnable := TRUE;
stXStage.bLimitBackwardEnable := TRUE;
stXStage.bHardwareEnable := TRUE;
stXStage.bPowerSelf := TRUE;

fbYStage(stMotionStage:=stYStage);
fbXStage(stMotionStage:=stXStage);

// We need to update from PLC or from EPICS, but not both
fbArrCheckWrite(
    astPositionState:=astPositionState,
    bCheck:=TRUE,
    bSave:=FALSE,
);
IF NOT fbArrCheckWrite.bHadWrite THEN
    astPositionState[E_TM2K2_States.OUT] := stOut;
    astPositionState[E_TM2K2_States.TARGET1] := stTarget1;
    astPositionState[E_TM2K2_States.TARGET2] := stTarget2;
    astPositionState[E_TM2K2_States.TARGET3] := stTarget3;
    astPositionState[E_TM2K2_States.TARGET4] := stTarget4;
    astPositionState[E_TM2K2_States.TARGET5] := stTarget5;
    astPositionState[E_TM2K2_States.TARGET6] := stTarget6;
END_IF

fbStates(
    stMotionStage:=stYStage,
    astPositionState:=astPositionState,
    eEnumSet:=eEnumSet,
    eEnumGet:=eEnumGet,
    fbFFHWO:=fbFFHWO,
    fbArbiter:=fbArbiter,
    bEnableMotion:=bEnableMotion,
    bEnableBeamParams:=bEnableBeamParams,
    bEnablePositionLimits:=bEnablePositionLimits,
    sDeviceName:=sDeviceName,
    sTransitionKey:=sTransitionKey,
    bReadDBNow:=bReadDBNow,
    stDbStateParams=>stDbStateParams,
);

fbArrCheckWrite(
    astPositionState:=astPositionState,
    bCheck:=FALSE,
    bSave:=TRUE,
);

stOut := astPositionState[E_TM2K2_States.OUT];
stTarget1 := astPositionState[E_TM2K2_States.TARGET1];
stTarget2 := astPositionState[E_TM2K2_States.TARGET2];
stTarget3 := astPositionState[E_TM2K2_States.TARGET3];
stTarget4 := astPositionState[E_TM2K2_States.TARGET4];
stTarget5 := astPositionState[E_TM2K2_States.TARGET5];
stTarget6 := astPositionState[E_TM2K2_States.TARGET6];

fbThermoCouple1();
fbFlowMeter();

END_FUNCTION_BLOCK

// ---- POUs/PRG_AT1K2_SOLID.TcPOU
PROGRAM PRG_AT1K2_SOLID
VAR
    (* NOTE: use FALSE for simulation and production *)
    (* NOTE: use TRUE when relying on visualization + actual hardware *)
    bDebug : BOOL := FALSE;

    nEnableMode : E_StageEnableMode;

    {attribute 'pytmc' := '
        pv: AT1K2:L2SI:MMS:01

    '}
    {attribute 'TcLinkTo' := '

        .fbRTD_1.iRaw := TIIB[AT1K2-EL3202-01]^RTD Inputs Channel 1^Value;
        .fbRTD_1.bError := TIIB[AT1K2-EL3202-01]^RTD Inputs Channel 1^Status^Error;
        .fbRTD_1.bUnderrange := TIIB[AT1K2-EL3202-01]^RTD Inputs Channel 1^Status^Underrange;
        .fbRTD_1.bOverrange := TIIB[AT1K2-EL3202-01]^RTD Inputs Channel 1^Status^Overrange;

        .fbRTD_2.iRaw := TIIB[AT1K2-EL3202-01]^RTD Inputs Channel 2^Value;
        .fbRTD_2.bError := TIIB[AT1K2-EL3202-01]^RTD Inputs Channel 2^Status^Error;
        .fbRTD_2.bUnderrange := TIIB[AT1K2-EL3202-01]^RTD Inputs Channel 2^Status^Underrange;
        .fbRTD_2.bOverrange := TIIB[AT1K2-EL3202-01]^RTD Inputs Channel 2^Status^Overrange

    '}
    fbStage1: FB_SXR_SATT_Stage;

    {attribute 'pytmc' := 'pv: AT1K2:L2SI:MMS:02'}
    {attribute 'TcLinkTo' := '

        .fbRTD_1.iRaw := TIIB[AT1K2-EL3202-02]^RTD Inputs Channel 1^Value;
        .fbRTD_1.bError := TIIB[AT1K2-EL3202-02]^RTD Inputs Channel 1^Status^Error;
        .fbRTD_1.bUnderrange := TIIB[AT1K2-EL3202-02]^RTD Inputs Channel 1^Status^Underrange;
        .fbRTD_1.bOverrange := TIIB[AT1K2-EL3202-02]^RTD Inputs Channel 1^Status^Overrange;

        .fbRTD_2.iRaw := TIIB[AT1K2-EL3202-02]^RTD Inputs Channel 2^Value;
        .fbRTD_2.bError := TIIB[AT1K2-EL3202-02]^RTD Inputs Channel 2^Status^Error;
        .fbRTD_2.bUnderrange := TIIB[AT1K2-EL3202-02]^RTD Inputs Channel 2^Status^Underrange;
        .fbRTD_2.bOverrange := TIIB[AT1K2-EL3202-02]^RTD Inputs Channel 2^Status^Overrange
    '}
    fbStage2: FB_SXR_SATT_Stage;

    // Special case: inspection mirror
    {attribute 'pytmc' := 'pv: AT1K2:L2SI:MMS:03'}
    fbStage3: FB_PositionState1D_InOut;
    bStage3Init: BOOL;
    fbMotionStage3: FB_MotionStage;
    stMirrorOut: ST_PositionState;
    stMirrorIn: ST_PositionState;
    // Consider transmission=1 if out, transmission=0 if in
    fMirrorTrans: LREAL;
    // Fault unless the mirror is out
    fbFFMirror: FB_FastFault := (
        i_Desc := 'Mirror is not out',
        i_TypeCode := E_MotionFFType.DEVICE_MOVE,
        i_xAutoReset := TRUE
    );

    fbStateSetup: FB_StateSetupHelper;
    stDefaultGood: ST_PositionState := (
        fDelta := 0.2,
        fVelocity := 1,
        bMoveOk := TRUE,
        bValid := TRUE
    );
    fbBadStateSetup: FB_StateSetupHelper;
    stDefaultBad: ST_PositionState := (
        fPosition := 500,
        fDelta := 0.2,
        fVelocity := 1,
        bMoveOk := FALSE,
        bValid := FALSE
    );

    {attribute 'pytmc' :='pv: AT1K2:L2SI:FWM'}
    {attribute 'TcLinkTo' := '.iRaw := TIIB[AT1K2-EL3052-E8]^AI Standard Channel 1^Value'}
    fbFlowMeter: FB_AnalogInput := (iTermBits:=15, fTermMax:=60, fTermMin:=0);

END_VAR

IF bDebug THEN
    // NEVER: checkouts with the TwinCAT NC GUI.
    nEnableMode := E_StageEnableMode.NEVER;
ELSE
    // ALWAYS: want active position correction at all times
    nEnableMode := E_StageEnableMode.ALWAYS;
END_IF

(*

    Solid Attenuator notes

    AT1K2 is JJ-xray SN-11343.

    JJ    Label   EPICS    Stage     NC   Location

    10XX      1   MMS:01   fbStage1  M25  Upstream-most
    10XX      2   MMS:02   fbStage2  M26  Downstream-most
    10XX      3   MMS:03   fbStage3  M27  Mirror Insertion Stage

*)

fbStateSetup(stPositionState:=stDefaultGood, bSetDefault:=TRUE);
fbBadStateSetup(stPositionState:=stDefaultBad, bSetDefault:=TRUE);


(* State setup - stage 1 *)
fbStateSetup(stPositionState:=fbStage1.stOut, sName:='Out', fPosition:=22.00);

fbBadStateSetup(stPositionState:=fbStage1.stFilter1, sName:='Filter 1',sPmpsState:='AT1K2:L2SI-RTD');
fbStage1.arrFilters[1].fFilterThickness_um := 0;
fbStage1.arrFilters[1].sFilterMaterial     := '';

fbBadStateSetup(stPositionState:=fbStage1.stFilter2, sName:='Filter 2');
fbStage1.arrFilters[2].fFilterThickness_um := 0;
fbStage1.arrFilters[2].sFilterMaterial     := '';

fbStateSetup(stPositionState:=fbStage1.stFilter3, sName:='(3) 11.5 um Al', fPosition:=75.0);
fbStage1.arrFilters[3].fFilterThickness_um := 11.5;
fbStage1.arrFilters[3].sFilterMaterial     := 'Al';

fbStateSetup(stPositionState:=fbStage1.stFilter4, sName:='(4) 6.18 um Al', fPosition:=90.5);
fbStage1.arrFilters[4].fFilterThickness_um := 6.18;
fbStage1.arrFilters[4].sFilterMaterial     := 'Al';

fbStateSetup(stPositionState:=fbStage1.stFilter5, sName:='(5) 2.85 um Al', fPosition:=105.5);
fbStage1.arrFilters[5].fFilterThickness_um := 2.85;
fbStage1.arrFilters[5].sFilterMaterial     := 'Al';

fbStateSetup(stPositionState:=fbStage1.stFilter6, sName:='(6) 1.52 um Al', fPosition:=122.0);
fbStage1.arrFilters[6].fFilterThickness_um := 1.52;
fbStage1.arrFilters[6].sFilterMaterial     := 'Al';

fbStateSetup(stPositionState:=fbStage1.stFilter7, sName:='(7) 0.78 um Al', fPosition:=136.5);
fbStage1.arrFilters[7].fFilterThickness_um := 0.78;
fbStage1.arrFilters[7].sFilterMaterial     := 'Al';

fbStateSetup(stPositionState:=fbStage1.stFilter8, sName:='(8) 0.39 um Al', fPosition:=152.2);
fbStage1.arrFilters[8].fFilterThickness_um := 0.39;
fbStage1.arrFilters[8].sFilterMaterial     := 'Al';

fbStage1 (stAxis:=Main.M25,sDeviceName:='AT1K2:L2SI', nEnableMode:=nEnableMode, fbFFHWO:=GVL.fbFastFaultOutput2, bEnable:=TRUE);


(* State setup - stage 2 *)
fbStateSetup(stPositionState:=fbStage2.stOut, sName:='Out', fPosition:=22.00);

fbBadStateSetup(stPositionState:=fbStage2.stFilter1, sName:='Filter 1',sPmpsState:='AT1K2:L2SI-RTD');
fbStage2.arrFilters[1].fFilterThickness_um := 0;
fbStage2.arrFilters[1].sFilterMaterial     := '';

fbBadStateSetup(stPositionState:=fbStage2.stFilter2, sName:='Filter 2');
fbStage2.arrFilters[2].fFilterThickness_um := 0;
fbStage2.arrFilters[2].sFilterMaterial     := '';

fbStateSetup(stPositionState:=fbStage2.stFilter3, sName:='(3) 11.5 um Al', fPosition:=75.0);
fbStage2.arrFilters[3].fFilterThickness_um := 11.5;
fbStage2.arrFilters[3].sFilterMaterial     := 'Al';

fbStateSetup(stPositionState:=fbStage2.stFilter4, sName:='(4) 6.18 um Al', fPosition:=90.5);
fbStage2.arrFilters[4].fFilterThickness_um := 6.18;
fbStage2.arrFilters[4].sFilterMaterial     := 'Al';

fbStateSetup(stPositionState:=fbStage2.stFilter5, sName:='(5) 1.52 um Al', fPosition:=105.5);
fbStage2.arrFilters[5].fFilterThickness_um := 1.52;
fbStage2.arrFilters[5].sFilterMaterial     := 'Al';

fbStateSetup(stPositionState:=fbStage2.stFilter6, sName:='(6) 0.78 um Al', fPosition:=122.0);
fbStage2.arrFilters[6].fFilterThickness_um := 0.78;
fbStage2.arrFilters[6].sFilterMaterial     := 'Al';

fbStateSetup(stPositionState:=fbStage2.stFilter7, sName:='(7) 0.39 um Al', fPosition:=136.5);
fbStage2.arrFilters[7].fFilterThickness_um := 0.39;
fbStage2.arrFilters[7].sFilterMaterial     := 'Al';

fbStateSetup(stPositionState:=fbStage2.stFilter8, sName:='(8) 0.2 um Al', fPosition:=152.2);
fbStage2.arrFilters[8].fFilterThickness_um := 0.2;
fbStage2.arrFilters[8].sFilterMaterial     := 'Al';

fbStage2(stAxis:=Main.M26,sDeviceName:='AT1K2:L2SI', nEnableMode:=nEnableMode, fbFFHWO:=GVL.fbFastFaultOutput2, bEnable:=TRUE);

(* State setup - stage 3 *)
fbStateSetup(stPositionState:=stMirrorOut, sName:='Out', fPosition:=65.00);
fbStateSetup(stPositionState:=stMirrorIn, sName:='In', fPosition:=25.00);

IF NOT bStage3Init THEN
    bStage3Init := TRUE;
    Main.M27.bHardwareEnable      := TRUE;
    Main.M27.bLimitBackwardEnable := TRUE;
    Main.M27.bLimitForwardEnable  := TRUE;
    Main.M27.bPowerSelf           := TRUE;
    Main.M27.nBrakeMode           := ENUM_StageBrakeMode.NO_BRAKE;
    Main.M27.nHomingMode          := ENUM_EpicsHomeCmd.NONE;
END_IF

fbStage3(
    stMotionStage:=Main.M27,
    stOut:=stMirrorOut,
    stIn:=stMirrorIn,
);
fbMotionStage3(stMotionStage:=Main.M27);

IF fbStage3.eStateGet = E_EpicsInOut.OUT THEN
    fMirrorTrans := 1.0;
ELSE
    fMirrorTrans := 0.0;
END_IF

fbFFMirror(
    i_DevName := Main.M27.sName,
    i_xOK := fbStage3.eStateGet = E_EpicsInOut.OUT,
    io_fbFFHWO := GVL.fbFastFaultOutput2,
);

GVL.rCurTrans[PMPS.K_Attenuators.AT1K2].nTran := LREAL_TO_REAL(
    fbStage1.fTransmission *
    fbStage2.fTransmission *
    fMirrorTrans
);

fbFlowMeter();

END_PROGRAM

// ---- POUs/PRG_AT2K2_SOLID.TcPOU
PROGRAM PRG_AT2K2_SOLID
VAR
    (* NOTE: use FALSE for simulation and production *)
    (* NOTE: use TRUE when relying on visualization + actual hardware *)
    bDebug : BOOL := FALSE;

    nEnableMode : E_StageEnableMode;

    {attribute 'pytmc' := '
        pv: AT2K2:L2SI:MMS:01

    '}
    {attribute 'TcLinkTo' := '

        .fbRTD_1.iRaw := TIIB[AT2K2-EL3202-04]^RTD Inputs Channel 1^Value;
        .fbRTD_1.bError := TIIB[AT2K2-EL3202-04]^RTD Inputs Channel 1^Status^Error;
        .fbRTD_1.bUnderrange := TIIB[AT2K2-EL3202-04]^RTD Inputs Channel 1^Status^Underrange;
        .fbRTD_1.bOverrange := TIIB[AT2K2-EL3202-04]^RTD Inputs Channel 1^Status^Overrange;

        .fbRTD_2.iRaw := TIIB[AT2K2-EL3202-04]^RTD Inputs Channel 2^Value;
        .fbRTD_2.bError := TIIB[AT2K2-EL3202-04]^RTD Inputs Channel 2^Status^Error;
        .fbRTD_2.bUnderrange := TIIB[AT2K2-EL3202-04]^RTD Inputs Channel 2^Status^Underrange;
        .fbRTD_2.bOverrange := TIIB[AT2K2-EL3202-04]^RTD Inputs Channel 2^Status^Overrange

    '}
    fbStage1: FB_SXR_SATT_Stage;

    {attribute 'pytmc' := 'pv: AT2K2:L2SI:MMS:02'}
    {attribute 'TcLinkTo' := '

        .fbRTD_1.iRaw := TIIB[AT2K2-EL3202-03]^RTD Inputs Channel 1^Value;
        .fbRTD_1.bError := TIIB[AT2K2-EL3202-03]^RTD Inputs Channel 1^Status^Error;
        .fbRTD_1.bUnderrange := TIIB[AT2K2-EL3202-03]^RTD Inputs Channel 1^Status^Underrange;
        .fbRTD_1.bOverrange := TIIB[AT2K2-EL3202-03]^RTD Inputs Channel 1^Status^Overrange;

        .fbRTD_2.iRaw := TIIB[AT2K2-EL3202-03]^RTD Inputs Channel 2^Value;
        .fbRTD_2.bError := TIIB[AT2K2-EL3202-03]^RTD Inputs Channel 2^Status^Error;
        .fbRTD_2.bUnderrange := TIIB[AT2K2-EL3202-03]^RTD Inputs Channel 2^Status^Underrange;
        .fbRTD_2.bOverrange := TIIB[AT2K2-EL3202-03]^RTD Inputs Channel 2^Status^Overrange

    '}
    fbStage2: FB_SXR_SATT_Stage;

    {attribute 'pytmc' := 'pv: AT2K2:L2SI:MMS:03'}
    {attribute 'TcLinkTo' := '

        .fbRTD_1.iRaw := TIIB[AT2K2-EL3202-02]^RTD Inputs Channel 1^Value;
        .fbRTD_1.bError := TIIB[AT2K2-EL3202-02]^RTD Inputs Channel 1^Status^Error;
        .fbRTD_1.bUnderrange := TIIB[AT2K2-EL3202-02]^RTD Inputs Channel 1^Status^Underrange;
        .fbRTD_1.bOverrange := TIIB[AT2K2-EL3202-02]^RTD Inputs Channel 1^Status^Overrange;

        .fbRTD_2.iRaw := TIIB[AT2K2-EL3202-02]^RTD Inputs Channel 2^Value;
        .fbRTD_2.bError := TIIB[AT2K2-EL3202-02]^RTD Inputs Channel 2^Status^Error;
        .fbRTD_2.bUnderrange := TIIB[AT2K2-EL3202-02]^RTD Inputs Channel 2^Status^Underrange;
        .fbRTD_2.bOverrange := TIIB[AT2K2-EL3202-02]^RTD Inputs Channel 2^Status^Overrange
    '}
    fbStage3: FB_SXR_SATT_Stage;

    {attribute 'pytmc' := 'pv: AT2K2:L2SI:MMS:04'}
    {attribute 'TcLinkTo' := '

        .fbRTD_1.iRaw := TIIB[AT2K2-EL3202-01]^RTD Inputs Channel 1^Value;
        .fbRTD_1.bError := TIIB[AT2K2-EL3202-01]^RTD Inputs Channel 1^Status^Error;
        .fbRTD_1.bUnderrange := TIIB[AT2K2-EL3202-01]^RTD Inputs Channel 1^Status^Underrange;
        .fbRTD_1.bOverrange := TIIB[AT2K2-EL3202-01]^RTD Inputs Channel 1^Status^Overrange;

        .fbRTD_2.iRaw := TIIB[AT2K2-EL3202-01]^RTD Inputs Channel 2^Value;
        .fbRTD_2.bError := TIIB[AT2K2-EL3202-01]^RTD Inputs Channel 2^Status^Error;
        .fbRTD_2.bUnderrange := TIIB[AT2K2-EL3202-01]^RTD Inputs Channel 2^Status^Underrange;
        .fbRTD_2.bOverrange := TIIB[AT2K2-EL3202-01]^RTD Inputs Channel 2^Status^Overrange
    '}
    fbStage4: FB_SXR_SATT_Stage;

    fbStateSetup: FB_StateSetupHelper;
    stDefaultGood: ST_PositionState := (
        fDelta := 0.2,
        fVelocity := 1,
        bMoveOk := TRUE,
        bValid := TRUE
    );
    fbBadStateSetup: FB_StateSetupHelper;
    stDefaultBad: ST_PositionState := (
        fPosition := 500,
        fDelta := 0.2,
        fVelocity := 1,
        bMoveOk := FALSE,
        bValid := FALSE
    );

    {attribute 'pytmc' :='pv: AT2K2:L2SI:FWM'}
    {attribute 'TcLinkTo' := '.iRaw := TIIB[TM2K2-EL3052-E6]^AI Standard Channel 1^Value'} // AT2K2 shares flow meter with TM2K2
    fbFlowMeter: FB_AnalogInput := (iTermBits:=15, fTermMax:=60, fTermMin:=0);
END_VAR



IF bDebug THEN
    // NEVER: checkouts with the TwinCAT NC GUI.
    nEnableMode := E_StageEnableMode.NEVER;
ELSE
    // ALWAYS: want active position correction at all times
    nEnableMode := E_StageEnableMode.ALWAYS;
END_IF

(*

    Solid Attenuator notes

    AT2K2 is JJ-xray SN-11343.

    JJ    Label   EPICS    Stage     NC   Location

    1087      1   MMS:01   fbStage1  M17  Upstream-most
    1088      2   MMS:02   fbStage2  M18
    1086      3   MMS:03   fbStage3  M19
    1089      4   MMS:04   fbStage4  M20  Downstream-most

*)

fbStateSetup(stPositionState:=stDefaultGood, bSetDefault:=TRUE);
fbBadStateSetup(stPositionState:=stDefaultBad, bSetDefault:=TRUE);


(* State setup - stage 1 *)
fbStateSetup(stPositionState:=fbStage1.stOut, sName:='Out', fPosition:=27.00);

fbBadStateSetup(stPositionState:=fbStage1.stFilter1, sName:='Filter 1',sPmpsState:='AT2K2:L2SI-RTD');
fbStage1.arrFilters[1].fFilterThickness_um := 0;
fbStage1.arrFilters[1].sFilterMaterial     := '';

fbBadStateSetup(stPositionState:=fbStage1.stFilter2, sName:='Filter 2');
fbStage1.arrFilters[2].fFilterThickness_um := 0;
fbStage1.arrFilters[2].sFilterMaterial     := '';

fbBadStateSetup(stPositionState:=fbStage1.stFilter3, sName:='Filter 3');
fbStage1.arrFilters[3].fFilterThickness_um := 0;
fbStage1.arrFilters[3].sFilterMaterial     := '';

fbBadStateSetup(stPositionState:=fbStage1.stFilter4, sName:='Filter 4');
fbStage1.arrFilters[4].fFilterThickness_um := 0;
fbStage1.arrFilters[4].sFilterMaterial     := '';

fbStateSetup(stPositionState:=fbStage1.stFilter5, sName:='(5) 11.5 um Al', fPosition:=103.0);
fbStage1.arrFilters[5].fFilterThickness_um := 11.5;
fbStage1.arrFilters[5].sFilterMaterial     := 'Al';

fbStateSetup(stPositionState:=fbStage1.stFilter6, sName:='(6) 6.18 um Al', fPosition:=119.0);
fbStage1.arrFilters[6].fFilterThickness_um := 6.18;
fbStage1.arrFilters[6].sFilterMaterial     := 'Al';

fbStateSetup(stPositionState:=fbStage1.stFilter7, sName:='(7) 2.85 um Al', fPosition:=135.0);
fbStage1.arrFilters[7].fFilterThickness_um := 2.85;
fbStage1.arrFilters[7].sFilterMaterial     := 'Al';

fbStateSetup(stPositionState:=fbStage1.stFilter8, sName:='(8) 1.52 um Al', fPosition:=150.0);
fbStage1.arrFilters[8].fFilterThickness_um := 1.52;
fbStage1.arrFilters[8].sFilterMaterial     := 'Al';

fbStage1(stAxis:=Main.M17,sDeviceName:='AT2K2:L2SI', nEnableMode:=nEnableMode, fbFFHWO:=GVL.fbFastFaultOutput2, bEnable:=TRUE);


(* State setup - stage 2 *)
fbStateSetup(stPositionState:=fbStage2.stOut, sName:='Out', fPosition:=27.72);

fbBadStateSetup(stPositionState:=fbStage2.stFilter1, sName:='Filter 1',sPmpsState:='AT2K2:L2SI-RTD');
fbStage2.arrFilters[1].fFilterThickness_um := 0;
fbStage2.arrFilters[1].sFilterMaterial     := '';

fbBadStateSetup(stPositionState:=fbStage2.stFilter2, sName:='Filter 2');
fbStage2.arrFilters[2].fFilterThickness_um := 0;
fbStage2.arrFilters[2].sFilterMaterial     := '';

fbBadStateSetup(stPositionState:=fbStage2.stFilter3, sName:='Filter 3');
fbStage2.arrFilters[3].fFilterThickness_um := 0;
fbStage2.arrFilters[3].sFilterMaterial     := '';

fbBadStateSetup(stPositionState:=fbStage2.stFilter4, sName:='Filter 4');
fbStage2.arrFilters[4].fFilterThickness_um := 0;
fbStage2.arrFilters[4].sFilterMaterial     := '';

fbStateSetup(stPositionState:=fbStage2.stFilter5, sName:='(5) 6.18 um Al', fPosition:=103.0);
fbStage2.arrFilters[5].fFilterThickness_um := 6.18;
fbStage2.arrFilters[5].sFilterMaterial     := 'Al';

fbStateSetup(stPositionState:=fbStage2.stFilter6, sName:='(6) 2.85 um Al', fPosition:=119.0);
fbStage2.arrFilters[6].fFilterThickness_um := 2.85;
fbStage2.arrFilters[6].sFilterMaterial     := 'Al';

fbStateSetup(stPositionState:=fbStage2.stFilter7, sName:='(7) 1.52 um Al', fPosition:=135.0);
fbStage2.arrFilters[7].fFilterThickness_um := 1.52;
fbStage2.arrFilters[7].sFilterMaterial     := 'Al';

fbStateSetup(stPositionState:=fbStage2.stFilter8, sName:='(8) 0.78 um Al', fPosition:=150.0);
fbStage2.arrFilters[8].fFilterThickness_um := 0.78;
fbStage2.arrFilters[8].sFilterMaterial     := 'Al';

fbStage2(stAxis:=Main.M18,sDeviceName:='AT2K2:L2SI', nEnableMode:=nEnableMode, fbFFHWO:=GVL.fbFastFaultOutput2, bEnable:=TRUE);


(* State setup - stage 3 *)
fbStateSetup(stPositionState:=fbStage3.stOut, sName:='Out', fPosition:=27.00);

fbBadStateSetup(stPositionState:=fbStage3.stFilter1, sName:='Filter 1',sPmpsState:='AT2K2:L2SI-RTD');
fbStage3.arrFilters[1].fFilterThickness_um := 0;
fbStage3.arrFilters[1].sFilterMaterial     := '';

fbBadStateSetup(stPositionState:=fbStage3.stFilter2, sName:='Filter 2');
fbStage3.arrFilters[2].fFilterThickness_um := 0;
fbStage3.arrFilters[2].sFilterMaterial     := '';

fbBadStateSetup(stPositionState:=fbStage3.stFilter3, sName:='Filter 3');
fbStage3.arrFilters[3].fFilterThickness_um := 0;
fbStage3.arrFilters[3].sFilterMaterial     := '';

fbBadStateSetup(stPositionState:=fbStage3.stFilter4, sName:='Filter 4');
fbStage3.arrFilters[4].fFilterThickness_um := 0;
fbStage3.arrFilters[4].sFilterMaterial     := '';

fbStateSetup(stPositionState:=fbStage3.stFilter5, sName:='(5) 2.85 um Al', fPosition:=103.0);
fbStage3.arrFilters[5].fFilterThickness_um := 2.85;
fbStage3.arrFilters[5].sFilterMaterial     := 'Al';

fbStateSetup(stPositionState:=fbStage3.stFilter6, sName:='(6) 1.52 um Al', fPosition:=119.0);
fbStage3.arrFilters[6].fFilterThickness_um := 1.52;
fbStage3.arrFilters[6].sFilterMaterial     := 'Al';

fbStateSetup(stPositionState:=fbStage3.stFilter7, sName:='(7) 0.78 um Al', fPosition:=135.0);
fbStage3.arrFilters[7].fFilterThickness_um := 0.78;
fbStage3.arrFilters[7].sFilterMaterial     := 'Al';

fbStateSetup(stPositionState:=fbStage3.stFilter8, sName:='(8) 0.39 um Al', fPosition:=150.0);
fbStage3.arrFilters[8].fFilterThickness_um := 0.39;
fbStage3.arrFilters[8].sFilterMaterial     := 'Al';

fbStage3(stAxis:=Main.M19,sDeviceName:='AT2K2:L2SI', nEnableMode:=nEnableMode, fbFFHWO:=GVL.fbFastFaultOutput2, bEnable:=TRUE);


(* State setup - stage 4 *)
fbStateSetup(stPositionState:=fbStage4.stOut, sName:='Out', fPosition:=28.03);

fbBadStateSetup(stPositionState:=fbStage4.stFilter1, sName:='Filter 1',sPmpsState:='AT2K2:L2SI-RTD');
fbStage4.arrFilters[1].fFilterThickness_um := 0;
fbStage4.arrFilters[1].sFilterMaterial     := '';

fbBadStateSetup(stPositionState:=fbStage4.stFilter2, sName:='Filter 2');
fbStage4.arrFilters[2].fFilterThickness_um := 0;
fbStage4.arrFilters[2].sFilterMaterial     := '';

fbBadStateSetup(stPositionState:=fbStage4.stFilter3, sName:='Filter 3');
fbStage4.arrFilters[3].fFilterThickness_um := 0;
fbStage4.arrFilters[3].sFilterMaterial     := '';

fbBadStateSetup(stPositionState:=fbStage4.stFilter4, sName:='Filter 4');
fbStage4.arrFilters[4].fFilterThickness_um := 0;
fbStage4.arrFilters[4].sFilterMaterial     := '';

fbStateSetup(stPositionState:=fbStage4.stFilter5, sName:='(5) 1.52 um Al', fPosition:=103.0);
fbStage4.arrFilters[5].fFilterThickness_um := 1.52;
fbStage4.arrFilters[5].sFilterMaterial     := 'Al';

fbStateSetup(stPositionState:=fbStage4.stFilter6, sName:='(6) 0.78 um Al', fPosition:=119.0);
fbStage4.arrFilters[6].fFilterThickness_um := 0.78;
fbStage4.arrFilters[6].sFilterMaterial     := 'Al';

fbStateSetup(stPositionState:=fbStage4.stFilter7, sName:='(7) 0.39 um Al', fPosition:=135.0);
fbStage4.arrFilters[7].fFilterThickness_um := 0.39;
fbStage4.arrFilters[7].sFilterMaterial     := 'Al';

fbStateSetup(stPositionState:=fbStage4.stFilter8, sName:='(8) 0.20 um Al', fPosition:=150.0);
fbStage4.arrFilters[8].fFilterThickness_um := 0.20;
fbStage4.arrFilters[8].sFilterMaterial     := 'Al';

fbStage4(stAxis:=Main.M20,sDeviceName:='AT2K2:L2SI', nEnableMode:=nEnableMode, fbFFHWO:=GVL.fbFastFaultOutput2, bEnable:=TRUE);


GVL.rCurTrans[PMPS.K_Attenuators.AT2K2].nTran := LREAL_TO_REAL(
    fbStage1.fTransmission *
    fbStage2.fTransmission *
    fbStage3.fTransmission *
    fbStage4.fTransmission
);

fbFlowMeter();

END_PROGRAM

// ---- POUs/PRG_LI3K2_K2B.TcPOU
PROGRAM PRG_LI3K2_K2B
VAR
    {attribute 'pytmc' := 'pv: LI3K2:K2B'}
    fbLI3K2: FB_LIC;

    fbStateSetup: FB_StateSetupHelper;
    stDefault: ST_PositionState := (
        fVelocity := 1,
        bMoveOk := TRUE,
        bValid := TRUE
    );
END_VAR


fbStateSetup(stPositionState:=stDefault, bSetDefault:=TRUE);

fbStateSetup(stPositionState:=fbLI3K2.stOut, fPosition:=0.118, sPmpsState:='LI3K2:K2B-OUT');
fbStateSetup(stPositionState:=fbLI3K2.stMirror1, fPosition:=-36.38, sPmpsState:='LI3K2:K2B-MIRROR1');
fbStateSetup(stPositionState:=fbLI3K2.stMirror2, fPosition:=-70.38, sPmpsState:='LI3K2:K2B-MIRROR2');
fbStateSetup(stPositionState:=fbLI3K2.stTarget1, fPosition:=-102.38, sPmpsState:='LI3K2:K2B-TARGET1');

fbLI3K2(
    fbFFHWO := GVL.fbFastFaultOutput2,
    fbArbiter := GVL.fbArbiter2,
    stYStage := Main.M21,
    sDeviceName := 'LI3K2:K2B',
    sTransitionKey := 'LI3K2:K2B-TRANSITION',
    bEnableMotion := TRUE,
    bEnableBeamParams := TRUE,
    bEnablePositionLimits := TRUE,
);

END_PROGRAM

// ---- POUs/PRG_PF2K2_WFS.TcPOU
PROGRAM PRG_PF2K2_WFS
VAR
    {attribute 'pytmc' := 'pv: PF2K2:WFS'}
    {attribute 'TcLinkTo' := '.fbThermoCouple1.bError 		:= TIIB[PF2K2-EL3314-E5]^TC Inputs Channel 1^Status^Error;
                              .fbThermoCouple1.bUnderrange	:= TIIB[PF2K2-EL3314-E5]^TC Inputs Channel 1^Status^Underrange;
                              .fbThermoCouple1.bOverrange 	:= TIIB[PF2K2-EL3314-E5]^TC Inputs Channel 1^Status^Overrange;
                              .fbThermoCouple1.iRaw 		:= TIIB[PF2K2-EL3314-E5]^TC Inputs Channel 1^Value;
                              .fbThermoCouple2.bError 		:= TIIB[PF2K2-EL3314-E5]^TC Inputs Channel 2^Status^Error;
                              .fbThermoCouple2.bUnderrange 	:= TIIB[PF2K2-EL3314-E5]^TC Inputs Channel 2^Status^Underrange;
                              .fbThermoCouple2.bOverrange 	:= TIIB[PF2K2-EL3314-E5]^TC Inputs Channel 2^Status^Overrange;
                              .fbThermoCouple2.iRaw 		:= TIIB[PF2K2-EL3314-E5]^TC Inputs Channel 2^Value'}
    fbPF2K2: FB_WFS;

    fbStateSetup: FB_StateSetupHelper;
    stDefault: ST_PositionState := (
        fVelocity := 1,
        bMoveOk := TRUE,
        bValid := TRUE
    );
END_VAR


fbStateSetup(stPositionState:=stDefault, bSetDefault:=TRUE);

fbStateSetup(stPositionState:=fbPF2K2.stOut, fPosition:=-15.00, sPmpsState:='PF2K2:WFS-OUT');
fbStateSetup(stPositionState:=fbPF2K2.stTarget1, fPosition:=-97.789, sPmpsState:='PF2K2:WFS-TARGET1');
fbStateSetup(stPositionState:=fbPF2K2.stTarget2, fPosition:=-83.416, sPmpsState:='PF2K2:WFS-TARGET2');
fbStateSetup(stPositionState:=fbPF2K2.stTarget3, fPosition:=-69.043, sPmpsState:='PF2K2:WFS-TARGET3');
fbStateSetup(stPositionState:=fbPF2K2.stTarget4, fPosition:=-54.669, sPmpsState:='PF2K2:WFS-TARGET4');
fbStateSetup(stPositionState:=fbPF2K2.stTarget5, fPosition:=-40.296, sPmpsState:='PF2K2:WFS-TARGET5');

fbPF2K2(
    fbFFHWO := GVL.fbFastFaultOutput2,
    fbArbiter := GVL.fbArbiter2,
    stYStage := Main.M22,
    stZStage := Main.M23,
    sDeviceName := 'PF2K2:WFS',
    sTransitionKey := 'PF2K2:WFS-TRANSITION',
    bEnableMotion := TRUE,
    bEnableBeamParams := TRUE,
    bEnablePositionLimits := TRUE,
    eEnumGet=>GVL.ePF2K2State,
);

END_PROGRAM

// ---- POUs/PRG_IM6K2_PPM.TcPOU
PROGRAM PRG_IM6K2_PPM
VAR
    {attribute 'pytmc' := 'pv: IM6K2:PPM'}
    {attribute 'TcLinkTo' := '.fbGige.iIlluminatorINT := TIIB[IM6K2-EL4004-E7]^AO Outputs Channel 1^Analog output;
                              .fbGige.bGigePower := TIIB[IM6K2-EL2004-E3]^Channel 2^Output;
                              .fbPowerMeter.iVoltageINT := TIIB[IM6K2-EL3602-E8]^AI Standard Channel 1^Value;
                              .fbPowerMeter.fbTempSensor.bError := TIIB[IM6K2-EL3314-E4]^TC Inputs Channel 1^Status^Error;
                              .fbPowerMeter.fbTempSensor.bUnderrange := TIIB[IM6K2-EL3314-E4]^TC Inputs Channel 1^Status^Underrange;
                              .fbPowerMeter.fbTempSensor.bOverrange := TIIB[IM6K2-EL3314-E4]^TC Inputs Channel 1^Status^Overrange;
                              .fbPowerMeter.fbTempSensor.iRaw := TIIB[IM6K2-EL3314-E4]^TC Inputs Channel 1^Value;
                              .fbYagTempSensor.bError := TIIB[IM6K2-EL3314-E4]^TC Inputs Channel 2^Status^Error;
                              .fbYagTempSensor.bUnderrange := TIIB[IM6K2-EL3314-E4]^TC Inputs Channel 2^Status^Underrange;
                              .fbYagTempSensor.bOverrange := TIIB[IM6K2-EL3314-E4]^TC Inputs Channel 2^Status^Overrange;
                              .fbYagTempSensor.iRaw := TIIB[IM6K2-EL3314-E4]^TC Inputs Channel 2^Value'}
    fbIM6K2: FB_PPM;

    fbStateSetup: FB_StateSetupHelper;
    stDefault: ST_PositionState := (
        fVelocity := 14,
        bMoveOk := TRUE,
        bValid := TRUE
    );
END_VAR


fbStateSetup(stPositionState:=stDefault, bSetDefault:=TRUE);

fbStateSetup(stPositionState:=fbIM6K2.stOut, fPosition:=-8.61, sPmpsState:='IM6K2:PPM-OUT');
fbStateSetup(stPositionState:=fbIM6K2.stPower, fPosition:=-47.71, sPmpsState:='IM6K2:PPM-POWERMETER');
fbStateSetup(stPositionState:=fbIM6K2.stYag1, fPosition:=-71.71);
fbStateSetup(stPositionState:=fbIM6K2.stYag2, fPosition:=-97.72, sPmpsState:='IM6K2:PPM-YAG2');

CASE GVL.ePF2K2State OF
    E_WFS_STATES.TARGET1, E_WFS_STATES.TARGET2, E_WFS_STATES.TARGET3, E_WFS_STATES.TARGET4, E_WFS_STATES.TARGET5 :
        // Known state targets: allow less strict pmps
        fbIM6K2.stYag1.stPMPS.sPmpsState := 'IM6K2:PPM-YAG1_WFS_IN';
ELSE
    // Out, Unknown, or an unexpected state: full pmps
    fbIM6K2.stYag1.stPMPS.sPmpsState := 'IM6K2:PPM-YAG1';
END_CASE

fbIM6K2(
    fbFFHWO := GVL.fbFastFaultOutput2,
    fbArbiter := GVL.fbArbiter2,
    stYStage := Main.M24,
    sDeviceName := 'IM6K2:PPM',
    sTransitionKey := 'IM6K2:PPM-TRANSITION',
    bEnableMotion := TRUE,
    bEnableBeamParams := TRUE,
    bEnablePositionLimits := TRUE,
    fResponsivity := 0.0719,
    iTermBits := 31,
    fTermMax := 1250,
    fTermMin := 0,
);

END_PROGRAM

// ---- POUs/PRG_SP1K2_PAX.TcPOU
PROGRAM PRG_SP1K2_PAX
VAR
    bInit : BOOL := TRUE;
    fbPAX_TAR_X : FB_MotionStage;
    fbPAX_TAR_Y : FB_MotionStage;
    fbPAX_TAR_Z : FB_MotionStage;

    fbPAX_BB_Y_01 : FB_MotionStage;
    fbPAX_BB_Y_02 : FB_MotionStage;

    fbPAX_FRAME_X : FB_MotionStage;
    fbPAX_FRAME_Y_01 : FB_MotionStage;
    fbPAX_FRAME_Y_02 : FB_MotionStage;
    fbPAX_FRAME_Y_03 : FB_MotionStage;

END_VAR

IF bInit THEN
    Main.M28.bHardwareEnable := TRUE;
    Main.M28.bPowerSelf := TRUE;

    Main.M29.bHardwareEnable := TRUE;
    Main.M29.bPowerSelf := TRUE;

    Main.M30.bHardwareEnable := TRUE;
    Main.M30.bPowerSelf := TRUE;

    Main.M31.bHardwareEnable := TRUE;
    Main.M31.bPowerSelf := TRUE;

    Main.M32.bHardwareEnable := TRUE;
    Main.M32.bPowerSelf := TRUE;

    Main.M33.bHardwareEnable := TRUE;
    Main.M33.bPowerSelf := TRUE;

    Main.M34.bHardwareEnable := TRUE;
    Main.M34.bPowerSelf := TRUE;

    Main.M36.bHardwareEnable := TRUE;
    Main.M36.bPowerSelf := TRUE;

    Main.M37.bHardwareEnable := TRUE;
    Main.M37.bPowerSelf := TRUE;

    bInit := FALSE;
END_IF

// PAX TAR
fbPAX_TAR_X(stMotionStage:= Main.M32);
fbPAX_TAR_Y(stMotionStage:= Main.M33);
fbPAX_TAR_Z(stMotionStage:= Main.M34);

// PAX BB
Main.M36.bLimitForwardEnable := TRUE;
Main.M36.bLimitBackwardEnable := TRUE;
fbPAX_BB_Y_01(stMotionStage:= Main.M36);

Main.M37.bLimitForwardEnable := TRUE;
Main.M37.bLimitBackwardEnable := TRUE;
fbPAX_BB_Y_02(stMotionStage:= Main.M37);

// FRAME
fbPAX_FRAME_X(stMotionStage:= Main.M31);
fbPAX_FRAME_Y_01(stMotionStage:= Main.M28);
fbPAX_FRAME_Y_02(stMotionStage:= Main.M29);
fbPAX_FRAME_Y_03(stMotionStage:= Main.M30);

END_PROGRAM

// ---- POUs/PRG_SP2K2_TXAS.TcPOU
PROGRAM PRG_SP2K2_TXAS
VAR
    bInit : BOOL := TRUE;
    fbTXAS_TAR_RX : FB_MotionStage;
    fbTXAS_YAG_FOCUS : FB_MotionStage;
END_VAR


IF bInit THEN
    Main.M38.bHardwareEnable := TRUE;
    Main.M38.bPowerSelf := TRUE;
    bInit := FALSE;

    Main.M41.bHardwareEnable := TRUE;
    Main.M41.bPowerSelf      := TRUE;
    Main.M41.fVelocity       := 0.1;
    Main.M41.nEnableMode     := E_StageEnableMode.DURING_MOTION;
    Main.M41.nBrakeMode      := E_StageBrakeMode.NO_BRAKE;
    Main.M41.nHomingMode     := E_EpicsHomeCmd.LOW_LIMIT;
    Main.M41.fHomePosition   := 0;
END_IF

Main.M38.bLimitBackwardEnable := TRUE;
Main.M38.bLimitForwardEnable := TRUE;

fbTXAS_TAR_RX(stMotionStage:=Main.M38);
fbTXAS_YAG_FOCUS(stMotionStage:=Main.M41);

END_PROGRAM

// ---- POUs/PRG_AT3K2_SOLID.TcPOU
PROGRAM PRG_AT3K2_SOLID
VAR
    bInit : BOOL := TRUE;
    bDebug : BOOL := FALSE;
    nEnableMode : E_StageEnableMode;

    {attribute 'pytmc' := 'pv: AT3K2:L2SI:MMS:01'}
    {attribute 'TcLinkTo' := '
        .fbRTD_1.iRaw := TIIB[K2S18-DRL-02-E9 (EL3202)]^RTD Inputs Channel 1^Value;
        .fbRTD_1.bError := TIIB[K2S18-DRL-02-E9 (EL3202)]^RTD Inputs Channel 1^Status^Error;
        .fbRTD_1.bUnderrange := TIIB[K2S18-DRL-02-E9 (EL3202)]^RTD Inputs Channel 1^Status^Underrange;
        .fbRTD_1.bOverrange := TIIB[K2S18-DRL-02-E9 (EL3202)]^RTD Inputs Channel 1^Status^Overrange;

        .fbRTD_2.iRaw := TIIB[K2S18-DRL-02-E9 (EL3202)]^RTD Inputs Channel 2^Value;
        .fbRTD_2.bError := TIIB[K2S18-DRL-02-E9 (EL3202)]^RTD Inputs Channel 2^Status^Error;
        .fbRTD_2.bUnderrange := TIIB[K2S18-DRL-02-E9 (EL3202)]^RTD Inputs Channel 2^Status^Underrange;
        .fbRTD_2.bOverrange := TIIB[K2S18-DRL-02-E9 (EL3202)]^RTD Inputs Channel 2^Status^Overrange

    '}
    fbStage1: FB_SXR_SATT_Stage;

    {attribute 'pytmc' := 'pv: AT3K2:L2SI:MMS:02'}
    {attribute 'TcLinkTo' := '

        .fbRTD_1.iRaw := TIIB[K2S18-DRL-02-E10 (EL3202)]^RTD Inputs Channel 1^Value;
        .fbRTD_1.bError := TIIB[K2S18-DRL-02-E10 (EL3202)]^RTD Inputs Channel 1^Status^Error;
        .fbRTD_1.bUnderrange := TIIB[K2S18-DRL-02-E10 (EL3202)]^RTD Inputs Channel 1^Status^Underrange;
        .fbRTD_1.bOverrange := TIIB[K2S18-DRL-02-E10 (EL3202)]^RTD Inputs Channel 1^Status^Overrange;

        .fbRTD_2.iRaw := TIIB[K2S18-DRL-02-E10 (EL3202)]^RTD Inputs Channel 2^Value;
        .fbRTD_2.bError := TIIB[K2S18-DRL-02-E10 (EL3202)]^RTD Inputs Channel 2^Status^Error;
        .fbRTD_2.bUnderrange := TIIB[K2S18-DRL-02-E10 (EL3202)]^RTD Inputs Channel 2^Status^Underrange;
        .fbRTD_2.bOverrange := TIIB[K2S18-DRL-02-E10 (EL3202)]^RTD Inputs Channel 2^Status^Overrange

    '}
    fbStage2: FB_SXR_SATT_Stage;

    fbStateSetup: FB_StateSetupHelper;
    stDefaultGood: ST_PositionState := (
        fDelta := 5,
        fVelocity := 1,
        bMoveOk := TRUE,
        bValid := TRUE
    );

    fbBadStateSetup: FB_StateSetupHelper;
    stDefaultBad: ST_PositionState := (
        fPosition := 500,
        fDelta := 0.2,
        fVelocity := 1,
        bMoveOk := FALSE,
        bValid := FALSE
    );
(*
    {attribute 'pytmc' :='pv: AT2K2:L2SI:FWM'}
    {attribute 'TcLinkTo' := '.iRaw := TIIB[TM2K2-EL3052-E6]^AI Standard Channel 1^Value'} // AT2K2 shares flow meter with TM2K2
    fbFlowMeter: FB_AnalogInput := (iTermBits:=15, fTermMax:=60, fTermMin:=0);
    *)
END_VAR

IF bDebug THEN
    // NEVER: checkouts with the TwinCAT NC GUI.
    nEnableMode := E_StageEnableMode.NEVER;
ELSE
    // ALWAYS: want active position correction at all times
    nEnableMode := E_StageEnableMode.ALWAYS;
END_IF

fbStateSetup(stPositionState:=stDefaultGood, bSetDefault:=TRUE);
fbBadStateSetup(stPositionState:=stDefaultBad, bSetDefault:=TRUE);


(* State setup - stage 1 *)
fbStateSetup(stPositionState:=fbStage1.stFilter8, sName:='1 um Co', fPosition:= 293, sPmpsState:='AT3K2:L2SI-RTD');
fbStage1.arrFilters[8].fFilterThickness_um := 1;
fbStage1.arrFilters[8].sFilterMaterial     := 'Co';

fbStateSetup(stPositionState:=fbStage1.stFilter7, sName:='2 um Co', fPosition:= 263);
fbStage1.arrFilters[7].fFilterThickness_um := 2;
fbStage1.arrFilters[7].sFilterMaterial     := 'Co';

fbStateSetup(stPositionState:=fbStage1.stFilter6, sName:='3 um Co', fposition:= 233);
fbStage1.arrFilters[6].fFilterThickness_um := 3;
fbStage1.arrFilters[6].sFilterMaterial     := 'Co';

fbStateSetup(stPositionState:=fbStage1.stFilter5, sName:='4 um Co', fPosition:= 173);
fbStage1.arrFilters[5].fFilterThickness_um := 4;
fbStage1.arrFilters[5].sFilterMaterial     := 'Co';

fbStateSetup(stPositionState:=fbStage1.stFilter4, sName:='5 um Co', fPosition:= 143);
fbStage1.arrFilters[4].fFilterThickness_um := 5;
fbStage1.arrFilters[4].sFilterMaterial     := 'Co';

fbStateSetup(stPositionState:=fbStage1.stFilter3, sName:='10 um Co', fPosition:= 180.0);
fbStage1.arrFilters[3].fFilterThickness_um := 10;
fbStage1.arrFilters[3].sFilterMaterial     := 'Al';

fbStateSetup(stPositionState:=fbStage1.stFilter2, sName:='15 um Co', fPosition:=113);
fbStage1.arrFilters[2].fFilterThickness_um := 15;
fbStage1.arrFilters[2].sFilterMaterial     := 'Al';

fbStateSetup(stPositionState:=fbStage1.stFilter1, sName:='20 um Co', fPosition:=83);
fbStage1.arrFilters[1].fFilterThickness_um := 20;
fbStage1.arrFilters[1].sFilterMaterial     := 'Al';

fbStateSetup(stPositionState:=fbStage1.stOut, sName:='Out', fPosition:=53);

fbStage1(stAxis:=Main.M39,sDeviceName:='AT3K2:L2SI', nEnableMode:=nEnableMode, fbFFHWO:=GVL.fbFastFaultOutput2, bEnable:=TRUE);


(* State setup - stage 2 *)

fbStateSetup(stPositionState:=fbStage2.stFilter8, sName:='0.2 um Co', fPosition:=265, sPmpsState:='AT3K2:L2SI-RTD');
fbStage2.arrFilters[8].fFilterThickness_um := 0.2;
fbStage2.arrFilters[8].sFilterMaterial     := 'Co';

fbStateSetup(stPositionState:=fbStage2.stFilter7, sName:='0.4 um Co', fPosition:= 235);
fbStage2.arrFilters[7].fFilterThickness_um := 0.4;
fbStage2.arrFilters[7].sFilterMaterial     := 'Co';

fbStateSetup(stPositionState:=fbStage2.stFilter6, sName:='0.6 um Co', fPosition:= 205);
fbStage2.arrFilters[6].fFilterThickness_um := 0.6;
fbStage2.arrFilters[6].sFilterMaterial     := 'Co';

fbStateSetup(stPositionState:=fbStage2.stFilter5, sName:='0.8 um Co', fPosition:= 175);
fbStage2.arrFilters[5].fFilterThickness_um := 0.8;
fbStage2.arrFilters[5].sFilterMaterial     := 'Co';

fbStateSetup(stPositionState:=fbStage2.stFilter4, sName:='1.0 um Co', fPosition:=145);
fbStage2.arrFilters[4].fFilterThickness_um := 1.0;
fbStage2.arrFilters[4].sFilterMaterial     := 'Co';

fbStateSetup(stPositionState:=fbStage2.stFilter3, sName:='1.5 um Co', fPosition:=115);
fbStage2.arrFilters[3].fFilterThickness_um := 1.5;
fbStage2.arrFilters[3].sFilterMaterial     := 'Co';

fbStateSetup(stPositionState:=fbStage2.stFilter2, sName:='2.0 um Co', fPosition:=85);
fbStage2.arrFilters[2].fFilterThickness_um := 2.0;
fbStage2.arrFilters[2].sFilterMaterial     := 'Co';

fbStateSetup(stPositionState:=fbStage2.stFilter1, sName:='3.0 um Co', fPosition:=55);
fbStage2.arrFilters[1].fFilterThickness_um := 3.0;
fbStage2.arrFilters[1].sFilterMaterial     := 'Al';

fbStateSetup(stPositionState:=fbStage2.stOut, sName:='Out', fPosition:=40.0);

fbStage2(stAxis:=Main.M40,sDeviceName:='AT3K2:L2SI', nEnableMode:=nEnableMode, fbFFHWO:=GVL.fbFastFaultOutput2, bEnable:=TRUE);

// GVL.rCurTrans[PMPS.K_Attenuators.AT2K2].nTran := LREAL_TO_REAL(
//PMPS.K_Attenuators.AT2K2; TODO: ADD TO ENUM?
GVL.rCurTrans[6].nTran := LREAL_TO_REAL(
    fbStage1.fTransmission *
    fbStage2.fTransmission
);

//fbFlowMeter();

END_PROGRAM

// ---- POUs/PRG_3_PMPS_POST.TcPOU
PROGRAM PRG_3_PMPS_POST
VAR
    fbArbiterIO: FB_SubSysToArbiter_IO;
    bMR1K1_Veto: BOOL;
    bST1K2_Veto: BOOL;
    bST1K2_Veto_Override: BOOL := FALSE;
    fb_vetoArbiter: FB_VetoArbiter;
    ff2_ff1_link_motion: FB_FastFault := (i_xAutoReset := TRUE, i_DevName := 'FF2 to FF1 Link Motion', i_Desc := 'Please DONT BYPASS ME!! This is virtual FF2 fault, Please check faulting motion devices', i_TypeCode := 16#FFFF);
END_VAR

bMR1K1_Veto := PMPS_GVL.stCurrentBeamParameters.aVetoDevices[PMPS.K_Stopper.MR1K1_OUT] AND NOT PMPS_GVL.stCurrentBeamParameters.aVetoDevices[PMPS.K_Stopper.MR1K1_IN];
bST1K2_Veto := bST1K2_Veto_Override OR PMPS_GVL.stCurrentBeamParameters.aVetoDevices[PMPS.K_Stopper.ST1K2];

fbArbiterIO(
    i_bVeto:=bMR1K1_Veto,
    Arbiter:=GVL.fbArbiter1,
    fbFFHWO:=GVL.fbFastFaultOutput1);

GVL.fbFastFaultOutput1.Execute(i_xVeto:=bMR1K1_Veto);
GVL.fbFastFaultOutput2.Execute(i_xVeto:=bMR1K1_Veto OR bST1K2_Veto);

//create a preemptive request from Arbiter 2 in Arbiter 1
fb_vetoArbiter(bVeto:= bST1K2_Veto,
                HigherAuthority := GVL.fbArbiter1,
                LowerAuthority := GVL.fbArbiter2,
                FFO := GVL.fbFastFaultOutput2);

ff2_ff1_link_motion(
    io_fbFFHWO := GVL.fbFastFaultOutput1,
    i_xOK :=  GVL.fbFastFaultOutput2.q_xFastFaultOut OR bST1K2_Veto);


MOTION_GVL.fbStandardPMPSDB(
    io_fbFFHWO:=GVL.fbFastFaultOutput1,
    bEnable:=TRUE,
    sPLCName:='plc-kfe-rix-motion',
);

END_PROGRAM

// ---- POUs/PRG_4_LOG.TcPOU
PROGRAM PRG_4_LOG
VAR
    fbLogHandler: FB_LogHandler;
END_VAR

fbLogHandler();

END_PROGRAM

// ---- POUs/PRG_ST3K2_TERM.TcPOU
PROGRAM PRG_ST3K2_TERM
VAR
    {attribute 'pytmc' := 'pv: ST3K2:TERM'}
    {attribute 'TcLinkTo' := 	'.i_xInsertedLS	:=	TIIB[ST3K2-TERM (EP2338-0001)]^Channel 4^Input;
                                 .i_xRetractedLS:=	TIIB[ST3K2-TERM (EP2338-0001)]^Channel 3^Input;
                                 .q_xRetract_DO	:=	TIIB[ST3K2-TERM (EP2338-0001)]^Channel 9^Output
    '}
    ST3K2: FB_MotionPneumaticActuator;
    ibPMPS_OK : BOOL;
END_VAR

ST3K2(
    ibInsertOK:= TRUE,
    ibRetractOK:= TRUE,
    ibPMPS_OK:= ibPMPS_OK,
    ibSingleCntrl:= TRUE ,
    ibCntrlHold:= TRUE,
    ibOverrideInterlock:= ,
    i_xReset:= ,
    stPneumaticActuator=> ,
    xMPS_OK=>  ,
    io_fbFFHWO:= GVL.fbFastFaultOutput2  );

END_PROGRAM
